VAR_OUTPUT
	EnO: BOOL;
	bDi_1: BOOL;
	bDi_2: BOOL;
	bDi_3: BOOL;
	bDi_4: BOOL;
	bDi_5: BOOL;
	bDi_6: BOOL;
	bDi_7: BOOL;
	bDi_8: BOOL;
	bDi_9: BOOL;
	bDi_10: BOOL;
	bDi_11: BOOL;
	bDi_12: BOOL;
	bDi_13: BOOL;
	bDi_14: BOOL;
	bDi_15: BOOL;
	bDi_16: BOOL;
	bError: BOOL;
END_VAR

VAR
	Channel_1_Input AT %I*: BOOL;
	Channel_2_Input AT %I*: BOOL;
	Channel_3_Input AT %I*: BOOL;
	Channel_4_Input AT %I*: BOOL;
	Channel_5_Input AT %I*: BOOL;
	Channel_6_Input AT %I*: BOOL;
	Channel_7_Input AT %I*: BOOL;
	Channel_8_Input AT %I*: BOOL;
	Channel_9_Input AT %I*: BOOL;
	Channel_10_Input AT %I*: BOOL;
	Channel_11_Input AT %I*: BOOL;
	Channel_12_Input AT %I*: BOOL;
	Channel_13_Input AT %I*: BOOL;
	Channel_14_Input AT %I*: BOOL;
	Channel_15_Input AT %I*: BOOL;
	Channel_16_Input AT %I*: BOOL;
	WcState_WcState AT %I*: BOOL;
	InfoData_State AT %I*: UINT;
	
	//FB-s
	EL1809_Error : FB_TerminalError;
END_VAR

EnO:=En;

//Error FB instance
EL1809_Error(
	En := TRUE,
	iTerminal_ID := iTerminal_ID,
	bWcState := WcState_WcState,
	uiInfoData_State := InfoData_State,
	pErrorSystem := ErrorSystem,
	bError => bError,
);

IF En THEN
	IF bError=FALSE THEN
		bDi_1:=Channel_1_Input;
		bDi_2:=Channel_2_Input;
		bDi_3:=Channel_3_Input;
		bDi_4:=Channel_4_Input;
		bDi_5:=Channel_5_Input;
		bDi_6:=Channel_6_Input;
		bDi_7:=Channel_7_Input;
		bDi_8:=Channel_8_Input;
		bDi_9:=Channel_9_Input;
		bDi_10:=Channel_10_Input;
		bDi_11:=Channel_11_Input;
		bDi_12:=Channel_12_Input;
		bDi_13:=Channel_13_Input;
		bDi_14:=Channel_14_Input;
		bDi_15:=Channel_15_Input;
		bDi_16:=Channel_16_Input;
	ELSE
		bDi_1:=FALSE;
		bDi_2:=FALSE;
		bDi_3:=FALSE;
		bDi_4:=FALSE;
		bDi_5:=FALSE;
		bDi_6:=FALSE;
		bDi_7:=FALSE;
		bDi_8:=FALSE;
		bDi_9:=FALSE;
		bDi_10:=FALSE;
		bDi_11:=FALSE;
		bDi_12:=FALSE;
		bDi_13:=FALSE;
		bDi_14:=FALSE;
		bDi_15:=FALSE;
		bDi_16:=FALSE;
	END_IF
END_IF

END_FUNCTION_BLOCK

// tc_mca_std_lib/POUs/Hardware/EtherCAT_Terminals/Digital_Inputs/EL1819
///EL1819 | HD EtherCAT Terminals, 16-channel digital input 24 V DC, 10 µs
FUNCTION_BLOCK EL1819

VAR_INPUT
	En: BOOL;
	iTerminal_ID : INT;
	ErrorSystem : POINTER TO ST_ErrorSystem;
END_VAR

VAR_OUTPUT
	EnO: BOOL;
	bDi_1: BOOL;
	bDi_2: BOOL;
	bDi_3: BOOL;
	bDi_4: BOOL;
	bDi_5: BOOL;
	bDi_6: BOOL;
	bDi_7: BOOL;
	bDi_8: BOOL;
	bDi_9: BOOL;
	bDi_10: BOOL;
	bDi_11: BOOL;
	bDi_12: BOOL;
	bDi_13: BOOL;
	bDi_14: BOOL;
	bDi_15: BOOL;
	bDi_16: BOOL;
	bError: BOOL;
END_VAR

VAR
	Channel_1_Input AT %I*: BOOL;
	Channel_2_Input AT %I*: BOOL;
	Channel_3_Input AT %I*: BOOL;
	Channel_4_Input AT %I*: BOOL;
	Channel_5_Input AT %I*: BOOL;
	Channel_6_Input AT %I*: BOOL;
	Channel_7_Input AT %I*: BOOL;
	Channel_8_Input AT %I*: BOOL;
	Channel_9_Input AT %I*: BOOL;
	Channel_10_Input AT %I*: BOOL;
	Channel_11_Input AT %I*: BOOL;
	Channel_12_Input AT %I*: BOOL;
	Channel_13_Input AT %I*: BOOL;
	Channel_14_Input AT %I*: BOOL;
	Channel_15_Input AT %I*: BOOL;
	Channel_16_Input AT %I*: BOOL;
	WcState_WcState AT %I*: BOOL;
	InfoData_State AT %I*: UINT;
	
	//FB-s
	EL1819_Error : FB_TerminalError;
END_VAR

EnO:=En;

//Error FB instance
EL1819_Error(
	En := TRUE,
	iTerminal_ID := iTerminal_ID,
	bWcState := WcState_WcState,
	uiInfoData_State := InfoData_State,
	pErrorSystem := ErrorSystem,
	bError => bError,
);

IF En THEN
	IF bError=FALSE THEN
		bDi_1:=Channel_1_Input;
		bDi_2:=Channel_2_Input;
		bDi_3:=Channel_3_Input;
		bDi_4:=Channel_4_Input;
		bDi_5:=Channel_5_Input;
		bDi_6:=Channel_6_Input;
		bDi_7:=Channel_7_Input;
		bDi_8:=Channel_8_Input;
		bDi_9:=Channel_9_Input;
		bDi_10:=Channel_10_Input;
		bDi_11:=Channel_11_Input;
		bDi_12:=Channel_12_Input;
		bDi_13:=Channel_13_Input;
		bDi_14:=Channel_14_Input;
		bDi_15:=Channel_15_Input;
		bDi_16:=Channel_16_Input;
	ELSE
		bDi_1:=FALSE;
		bDi_2:=FALSE;
		bDi_3:=FALSE;
		bDi_4:=FALSE;
		bDi_5:=FALSE;
		bDi_6:=FALSE;
		bDi_7:=FALSE;
		bDi_8:=FALSE;
		bDi_9:=FALSE;
		bDi_10:=FALSE;
		bDi_11:=FALSE;
		bDi_12:=FALSE;
		bDi_13:=FALSE;
		bDi_14:=FALSE;
		bDi_15:=FALSE;
		bDi_16:=FALSE;
	END_IF
END_IF

END_FUNCTION_BLOCK

// tc_mca_std_lib/POUs/Hardware/EtherCAT_Terminals/Digital_Inputs/FB_EL1252ASM_v1_00
FUNCTION_BLOCK FB_EL1252ASM_v1_00
VAR_INPUT
	En: BOOL;
END_VAR
VAR_OUTPUT
	EnO: BOOL;
	Di_1: BOOL;
	Di_2: BOOL;
	Di_1_LatchTimePos: ULINT;
	Di_2_LatchTimePos: ULINT;
	Di_1_LatchTimeNeg: ULINT;
	Di_2_LatchTimeNeg: ULINT;
	///Below bits can be used but then they must be enabled in the COE of the card. Nicklas suggested to not use these (since something wss written that you then only were allowed to read the latch time onece (some kkind of auto reset??))	
	///Di_1_LatchNeg:BOOL;
	///	Di_1_LatchPos:BOOL;
	///	Di_2_LatchNeg:BOOL;
	///	Di_2_LatchPos:BOOL;
	Error: BOOL;
END_VAR
VAR
	Channel_1_Input AT %I*: BOOL;
	Channel_2_Input AT %I*: BOOL;
	///Latch_Status1 AT %I*: USINT;
	///	Latch_Status2 AT %I*: USINT;
	Latch_LatchPos1 AT %I*: ULINT;
	Latch_LatchNeg1 AT %I*: ULINT;
	Latch_LatchPos2 AT %I*: ULINT;
	Latch_LatchNeg2 AT %I*: ULINT;
	WcState_WcState AT %I*: BOOL;
	InfoData_State AT %I*: UINT;
END_VAR

EnO:=En;

IF En AND (WcState_WcState OR InfoData_State<>16#8) THEN //InfoData_State==0 => in OP mode
	Error:=TRUE;
ELSE
	Error:=FALSE;
END_IF

IF En THEN
	IF Error=FALSE THEN
		Di_1:=Channel_1_Input;
		Di_2:=Channel_2_Input;
	(*	Di_1_LatchPos:=Latch_Status1.0;
		Di_1_LatchNeg:=Latch_Status1.1;
		Di_2_LatchPos:=Latch_Status2.0;
		Di_2_LatchNeg:=Latch_Status2.1;*)
		Di_1_LatchTimePos:=Latch_LatchPos1;
		Di_2_LatchTimePos:=Latch_LatchPos2;		
		Di_1_LatchTimeNeg:=Latch_LatchNeg1;		
		Di_2_LatchTimeNeg:=Latch_LatchNeg2;
		
	ELSE
		Di_1:=FALSE;
		Di_2:=FALSE;
	END_IF
END_IF

END_FUNCTION_BLOCK

// tc_mca_std_lib/POUs/Hardware/EtherCAT_Terminals/Digital_Outputs/EL2014
FUNCTION_BLOCK EL2014
VAR_INPUT
	En: BOOL;
	iTerminal_ID : INT; 
	bDo_1: BOOL;
	bDo_2: BOOL;
	bDo_3: BOOL;
	bDo_4: BOOL;
	ErrorSystem : POINTER TO ST_ErrorSystem;
END_VAR

VAR_OUTPUT
	EnO : BOOL;
	bError : BOOL;
END_VAR

VAR
	Channel_1_Output AT %Q*: BOOL;
	Channel_2_Output AT %Q*: BOOL;
	Channel_3_Output AT %Q*: BOOL;
	Channel_4_Output AT %Q*: BOOL;
	WcState_WcState AT %I*: BOOL;
	InfoData_State AT %I*: UINT;
	
	//FB-s
	EL2014_Error : FB_TerminalError;
END_VAR

(*
* TODO:
* Channel diagnostic variables and device diag variables
*)

EnO:=En;

EL2014_Error(
	En := TRUE,
	iTerminal_ID := iTerminal_ID,
	bWcState := WcState_WcState,
	uiInfoData_State := InfoData_State,
	pErrorSystem := ErrorSystem,
	bError => bError,
);

IF En THEN
	IF bError=FALSE THEN
		Channel_1_Output:=bDo_1;
		Channel_2_Output:=bDo_2;
		Channel_3_Output:=bDo_3;
		Channel_4_Output:=bDo_4;
	ELSE
		Channel_1_Output:=FALSE;
		Channel_2_Output:=FALSE;
		Channel_3_Output:=FALSE;
		Channel_4_Output:=FALSE;
	END_IF
END_IF

END_FUNCTION_BLOCK

// tc_mca_std_lib/POUs/Hardware/EtherCAT_Terminals/Digital_Outputs/EL2252
///EL2252 | XFC, 2-channel digital output terminal with time stamp, tri-state
FUNCTION_BLOCK EL2252
VAR_INPUT
	En: BOOL;
	iTerminal_ID : INT; 
	bDo_1: BOOL;
	bDo_2: BOOL;
ErrorSystem : POINTER TO ST_ErrorSystem;
END_VAR

VAR_OUTPUT
	EnO : BOOL;
	bError : BOOL;
END_VAR

VAR
	Channel_1_Output AT %Q*: BOOL;
	Channel_2_Output AT %Q*: BOOL;
	WcState_WcState AT %I*: BOOL;
	InfoData_State AT %I*: UINT;
	
	//FB-s
	EL2252_Error : FB_TerminalError;
END_VAR

(*
* TODO:
* Add the DC sync variables
*)

EL2252_Error(
	En := TRUE,
	iTerminal_ID := iTerminal_ID,
	bWcState := WcState_WcState,
	uiInfoData_State := InfoData_State,
	pErrorSystem := ErrorSystem,
	bError => bError,
);

IF En THEN
	IF bError=FALSE THEN
		Channel_1_Output:=bDo_1;
		Channel_2_Output:=bDo_2;
	ELSE
		Channel_1_Output:=FALSE;
		Channel_2_Output:=FALSE;
	END_IF
END_IF

END_FUNCTION_BLOCK

// tc_mca_std_lib/POUs/Hardware/EtherCAT_Terminals/Digital_Outputs/EL2808
FUNCTION_BLOCK EL2808

VAR_INPUT
	En: BOOL;
	iTerminal_ID : INT; 
	bDo_1: BOOL;
	bDo_2: BOOL;
	bDo_3: BOOL;
	bDo_4: BOOL;
	bDo_5: BOOL;
	bDo_6: BOOL;
	bDo_7: BOOL;
	bDo_8: BOOL;
	ErrorSystem : POINTER TO ST_ErrorSystem;
END_VAR

VAR_OUTPUT
	EnO : BOOL;
	bError : BOOL;
END_VAR

VAR
	Channel_1_Output AT %Q*: BOOL;
	Channel_2_Output AT %Q*: BOOL;
	Channel_3_Output AT %Q*: BOOL;
	Channel_4_Output AT %Q*: BOOL;
	Channel_5_Output AT %Q*: BOOL;
	Channel_6_Output AT %Q*: BOOL;
	Channel_7_Output AT %Q*: BOOL;
	Channel_8_Output AT %Q*: BOOL;
	WcState_WcState AT %I*: BOOL;
	InfoData_State AT %I*: UINT;
	
	//FB-s
	EL2808_Error : FB_TerminalError;
END_VAR

EnO:=En;

EL2808_Error(
	En := TRUE,
	iTerminal_ID := iTerminal_ID,
	bWcState := WcState_WcState,
	uiInfoData_State := InfoData_State,
	pErrorSystem := ErrorSystem,
	bError => bError,
);

IF En THEN
	IF bError=FALSE THEN
		Channel_1_Output:=bDo_1;
		Channel_2_Output:=bDo_2;
		Channel_3_Output:=bDo_3;
		Channel_4_Output:=bDo_4;
		Channel_5_Output:=bDo_5;
		Channel_6_Output:=bDo_6;
		Channel_7_Output:=bDo_7;
		Channel_8_Output:=bDo_8;
	ELSE
		Channel_1_Output:=FALSE;
		Channel_2_Output:=FALSE;
		Channel_3_Output:=FALSE;
		Channel_4_Output:=FALSE;
		Channel_5_Output:=FALSE;
		Channel_6_Output:=FALSE;
		Channel_7_Output:=FALSE;
		Channel_8_Output:=FALSE;
	END_IF
END_IF

END_FUNCTION_BLOCK

// tc_mca_std_lib/POUs/Hardware/EtherCAT_Terminals/Digital_Outputs/EL2819
FUNCTION_BLOCK EL2819
VAR_INPUT
	En: BOOL;
	iTerminal_ID : INT; 
	bDo_1: BOOL;
	bDo_2: BOOL;
	bDo_3: BOOL;
	bDo_4: BOOL;
	bDo_5: BOOL;
	bDo_6: BOOL;
	bDo_7: BOOL;
	bDo_8: BOOL;
	bDo_9: BOOL;
	bDo_10: BOOL;
	bDo_11: BOOL;
	bDo_12: BOOL;
	bDo_13: BOOL;
	bDo_14: BOOL;
	bDo_15: BOOL;
	bDo_16: BOOL;
	ErrorSystem : POINTER TO ST_ErrorSystem;
END_VAR

VAR_OUTPUT
	EnO : BOOL;
	bError : BOOL;
END_VAR

VAR
	Channel_1_Output AT %Q*: BOOL;
	Channel_2_Output AT %Q*: BOOL;
	Channel_3_Output AT %Q*: BOOL;
	Channel_4_Output AT %Q*: BOOL;
	Channel_5_Output AT %Q*: BOOL;
	Channel_6_Output AT %Q*: BOOL;
	Channel_7_Output AT %Q*: BOOL;
	Channel_8_Output AT %Q*: BOOL;
	Channel_9_Output AT %Q*: BOOL;
	Channel_10_Output AT %Q*: BOOL;
	Channel_11_Output AT %Q*: BOOL;
	Channel_12_Output AT %Q*: BOOL;
	Channel_13_Output AT %Q*: BOOL;
	Channel_14_Output AT %Q*: BOOL;
	Channel_15_Output AT %Q*: BOOL;
	Channel_16_Output AT %Q*: BOOL;
	
	WcState_WcState AT %I*: BOOL;
	InfoData_State AT %I*: UINT;
	
	//FB-s
	EL2819_Error : FB_TerminalError;
END_VAR

(*
* TODO:
* Channel diagnostic variables and device diag variables
*)

EnO:=En;

EL2819_Error(
	En := TRUE,
	iTerminal_ID := iTerminal_ID,
	bWcState := WcState_WcState,
	uiInfoData_State := InfoData_State,
	pErrorSystem := ErrorSystem,
	bError => bError,
);

IF En THEN
	IF bError=FALSE THEN
		Channel_1_Output:=bDo_1;
		Channel_2_Output:=bDo_2;
		Channel_3_Output:=bDo_3;
		Channel_4_Output:=bDo_4;
		Channel_5_Output:=bDo_5;
		Channel_6_Output:=bDo_6;
		Channel_7_Output:=bDo_7;
		Channel_8_Output:=bDo_8;
		Channel_9_Output:=bDo_9;
		Channel_10_Output:=bDo_10;
		Channel_11_Output:=bDo_11;
		Channel_12_Output:=bDo_12;
		Channel_13_Output:=bDo_13;
		Channel_14_Output:=bDo_14;
		Channel_15_Output:=bDo_15;
		Channel_16_Output:=bDo_16;
	ELSE
		Channel_1_Output:=FALSE;
		Channel_2_Output:=FALSE;
		Channel_3_Output:=FALSE;
		Channel_4_Output:=FALSE;
		Channel_5_Output:=FALSE;
		Channel_6_Output:=FALSE;
		Channel_7_Output:=FALSE;
		Channel_8_Output:=FALSE;
		Channel_9_Output:=FALSE;
		Channel_10_Output:=FALSE;
		Channel_11_Output:=FALSE;
		Channel_12_Output:=FALSE;
		Channel_13_Output:=FALSE;
		Channel_14_Output:=FALSE;
		Channel_15_Output:=FALSE;
		Channel_16_Output:=FALSE;
	END_IF
END_IF

END_FUNCTION_BLOCK

// tc_mca_std_lib/POUs/Hardware/EtherCAT_Terminals/Measuring_Terminals/EL5002
//EL5002 | 2-chennel SSI absolute encoder terminal
FUNCTION_BLOCK EL5002

VAR_INPUT
	En: BOOL;
	iTerminal_ID : INT;
	ErrorSystem : POINTER TO ST_ErrorSystem;
END_VAR

VAR_OUTPUT
	EnO: BOOL;
	Ch1_Counter_Value : UDINT;
	Ch2_Counter_Value : UDINT;
	bError: BOOL;
END_VAR

VAR
	udi_Ch1_Cnt_Value AT %I* : UDINT;
	udi_Ch2_Cnt_Value AT %I* : UDINT;
	WcState_WcState AT %I*: BOOL;
	InfoData_State AT %I*: UINT;
	
	//FB-s
	EL5002_Error : FB_TerminalError;
END_VAR

(*
* TODO:
* Channel Status words
*)

EnO:=En;

//Error FB instance
EL5002_Error(
	En := TRUE,
	iTerminal_ID := iTerminal_ID,
	bWcState := WcState_WcState,
	uiInfoData_State := InfoData_State,
	pErrorSystem := ErrorSystem,
	bError => bError,
);

IF EN THEN
	IF NOT bError THEN
		Ch1_Counter_Value := udi_Ch1_Cnt_Value;
		Ch2_Counter_Value := udi_Ch2_Cnt_Value;
	ELSE
		Ch1_Counter_Value := 0;
		Ch2_Counter_Value := 0;
	END_IF
END_IF

END_FUNCTION_BLOCK

// tc_mca_std_lib/POUs/Hardware/EtherCAT_Terminals/Measuring_Terminals/EL5021
//EL5021 | 1-channel Sin/Cos encoder
FUNCTION_BLOCK EL5021

VAR_INPUT
	En: BOOL;
	iTerminal_ID : INT;
	ErrorSystem : POINTER TO ST_ErrorSystem;
END_VAR

VAR_OUTPUT
	EnO: BOOL;
	Counter_Value : UDINT;
	Latch_Value : UDINT;
	bError: BOOL;
END_VAR

VAR
	udiCounter_Value AT %I* : UDINT;
	udiLatch_Value AT %I* : UDINT;
	WcState_WcState AT %I*: BOOL;
	InfoData_State AT %I*: UINT;
	
	//FB-s
	EL5021_Error : FB_TerminalError;
END_VAR

(*
* TODO:
* Channel Status words, control words
*)

EnO:=En;

//Error FB instance
EL5021_Error(
	En := TRUE,
	iTerminal_ID := iTerminal_ID,
	bWcState := WcState_WcState,
	uiInfoData_State := InfoData_State,
	pErrorSystem := ErrorSystem,
	bError => bError,
);

IF EN THEN
	IF NOT bError THEN
		Counter_Value := udiCounter_Value;
		Latch_Value := udiLatch_Value;
	ELSE
		Counter_Value := 0;
		Latch_Value := 0;
	END_IF
END_IF

END_FUNCTION_BLOCK

// tc_mca_std_lib/POUs/Hardware/EtherCAT_Terminals/Measuring_Terminals/EL5042
//EL5042 | 2-channel BiSS-C absolute encoder terminal
FUNCTION_BLOCK EL5042

VAR_INPUT
	En: BOOL;
	iTerminal_ID : INT;
	ErrorSystem : POINTER TO ST_ErrorSystem;
END_VAR

VAR_OUTPUT
	EnO: BOOL;
	Ch1_Position : ULINT;
	Ch2_Position : ULINT;
	bError: BOOL;
END_VAR

VAR
	FB_Inputs_ch1_Position AT %I* : ULINT;
	FB_Inputs_ch2_Position AT %I* : ULINT;
	WcState_WcState AT %I*: BOOL;
	InfoData_State AT %I*: UINT;
	
	//FB-s
	EL5042_Error : FB_TerminalError;
END_VAR

(*
* TODO:
* Channel Status words
*)

EnO:=En;

//Error FB instance
EL5042_Error(
	En := TRUE,
	iTerminal_ID := iTerminal_ID,
	bWcState := WcState_WcState,
	uiInfoData_State := InfoData_State,
	pErrorSystem := ErrorSystem,
	bError => bError,
);

IF EN THEN
	IF NOT bError THEN
		Ch1_Position := FB_Inputs_ch1_Position;
		Ch2_Position := FB_Inputs_ch2_Position;
	ELSE
		Ch1_Position := 0;
		Ch2_Position := 0;
	END_IF
END_IF

END_FUNCTION_BLOCK

// tc_mca_std_lib/POUs/Hardware/EtherCAT_Terminals/Measuring_Terminals/EL5101
// EL5101 | 1-channel incremental encoder terminal, 5V, RS422
FUNCTION_BLOCK EL5101

VAR_INPUT
	En: BOOL;
	iTerminal_ID : INT;
	ErrorSystem : POINTER TO ST_ErrorSystem;
END_VAR

VAR_OUTPUT
	EnO: BOOL;
	Counter_Value : UINT;
	Latch_Value : UINT;
	bError: BOOL;
END_VAR

VAR
	uiCounter_Value AT %I* : UINT;
	uiLatch_Value AT %I* : UINT;
	WcState_WcState AT %I*: BOOL;
	InfoData_State AT %I*: UINT;
	
	//FB-s
	EL5101_Error : FB_TerminalError;
END_VAR

(*
* TODO:
* Channel Status word, control words
*)

EnO:=En;

//Error FB instance
EL5101_Error(
	En := TRUE,
	iTerminal_ID := iTerminal_ID,
	bWcState := WcState_WcState,
	uiInfoData_State := InfoData_State,
	pErrorSystem := ErrorSystem,
	bError => bError,
);

IF EN THEN
	IF NOT bError THEN
		Counter_Value := uiCounter_Value;
		Latch_Value := uiLatch_Value;
	ELSE
		Counter_Value := 0;
		Latch_Value := 0;
	END_IF
END_IF

END_FUNCTION_BLOCK

// tc_mca_std_lib/POUs/Hardware/EtherCAT_Terminals/Motion/EL7211_v1_00
///EL7211 | Servo motor termional 5 A
FUNCTION_BLOCK EL7211_v1_00
VAR_INPUT
	En: BOOL;
END_VAR
VAR_OUTPUT
	EnO: BOOL;

	bError: BOOL;
END_VAR
VAR
	WcState_WcState AT %I*: BOOL;
	InfoData_State AT %I*: UINT;
END_VAR

EnO:=En;

IF En AND (WcState_WcState OR InfoData_State<>16#8) THEN
	bError:=TRUE;
ELSE
	bError:=FALSE;
END_IF

END_FUNCTION_BLOCK

// tc_mca_std_lib/POUs/Hardware/EtherCAT_Terminals/Motion/EL9576_v1_00
///EL9576 | Brake terminal (vap and resistor)
FUNCTION_BLOCK EL9576_v1_00
VAR_INPUT
	En: BOOL;
END_VAR
VAR_OUTPUT
	EnO: BOOL;
	bError: BOOL;	
	OverTemperature: BOOL;
	I2TError : BOOL;
	I2TWarning : BOOL;
	OverVoltage  : BOOL;
	UnderVoltage : BOOL;
	ChopperOn : BOOL;
	DCLinkVoltage : LREAL;
	DutyCycle  : LREAL;
	ResistorCurrent : LREAL;
	
END_VAR
VAR
	BCTOverTemperature AT %I*: BOOL;
	BCTI2TError AT %I*: BOOL;
	BCTI2TWarning AT %I*: BOOL;
	BCTOverVoltage  AT %I*: BOOL;
	BCTUnderVoltage  AT %I*: BOOL;
	BCTChopperOn  AT %I*: BOOL;
	BCTDCLinkVoltage AT %I*: UDINT;
	BCTDutyCycle  AT %I*: USINT;
	BCTResistorCurrent AT %I*: UDINT;
	WcState_WcState AT %I*: BOOL;
	InfoData_State AT %I*: UINT;
	
END_VAR

EnO:=En;

IF En AND (WcState_WcState OR InfoData_State<>16#8 OR BCTI2TError OR BCTI2TWarning OR BCTOverTemperature OR BCTOverVoltage OR BCTUnderVoltage) THEN
	bError:=TRUE;
ELSE
	bError:=FALSE;
END_IF

OverTemperature:=BCTOverTemperature;
I2TError:=BCTI2TError;
I2TWarning:=BCTI2TWarning;
OverVoltage:=BCTOverVoltage;
UnderVoltage:=bctUnderVoltage;
ChopperOn:=bctChopperOn;
DCLinkVoltage:=UDINT_TO_LREAL(bctDCLinkVoltage);
DutyCycle:=USINT_TO_LREAL(BCTDutyCycle);
ResistorCurrent:=UDINT_TO_LREAL(BCTResistorCurrent);

END_FUNCTION_BLOCK

// tc_mca_std_lib/POUs/Hardware/EtherCAT_Terminals/System/EL9410
//EL9410 | E-Bus power supplier and refresher, diagnostics
FUNCTION_BLOCK EL9410

VAR_INPUT
	En: BOOL;
	iTerminal_ID : INT;
	ErrorSystem : POINTER TO ST_ErrorSystem;
END_VAR

VAR_OUTPUT
	EnO: BOOL;
	bError: BOOL;
END_VAR

VAR
	bStatus_Us_UV AT %I* : BOOL;
	bStatus_Up_UV AT %I* : BOOL;
	WcState_WcState AT %I*: BOOL;
	InfoData_State AT %I*: UINT;
	
	//FB-s
	EL9410_Error : FB_TerminalError;
END_VAR

(*
* TODO:
* Status bits
*)

EnO:=En;

//Error FB instance
EL9410_Error(
	En := TRUE,
	iTerminal_ID := iTerminal_ID,
	bWcState := WcState_WcState,
	uiInfoData_State := InfoData_State,
	pErrorSystem := ErrorSystem,
	bError => bError,
);

END_FUNCTION_BLOCK

// tc_mca_std_lib/POUs/Hardware/EtherCAT_Terminals/System/EL9505
//EL9505 | Power supply terminal 5V
FUNCTION_BLOCK EL9505

VAR_INPUT
	En: BOOL;
	iTerminal_ID : INT;
	ErrorSystem : POINTER TO ST_ErrorSystem;
END_VAR

VAR_OUTPUT
	EnO: BOOL;
	bError: BOOL;
END_VAR

VAR
	bStatus_Uo_Power_OK AT %I* : BOOL;
	bStatus_Uo_Overload AT %I* : BOOL;
	WcState_WcState AT %I*: BOOL;
	InfoData_State AT %I*: UINT;
	
	//FB-s
	EL9505_Error : FB_TerminalError;
END_VAR

(*
* TODO:
* Status bits
*)
EnO:=En;

//Error FB instance
EL9505_Error(
	En := TRUE,
	iTerminal_ID := iTerminal_ID,
	bWcState := WcState_WcState,
	uiInfoData_State := InfoData_State,
	pErrorSystem := ErrorSystem,
	bError => bError,
);

END_FUNCTION_BLOCK

// tc_mca_std_lib/POUs/Hardware/Other/EK1200
FUNCTION_BLOCK EK1200
VAR_INPUT
	En: BOOL;
END_VAR
VAR_OUTPUT
	EnO: BOOL;
END_VAR

EnO:=En;

END_FUNCTION_BLOCK

// tc_mca_std_lib/POUs/Motion/FB_NcAxis
///#########################################################
///Function block to communicate between Nc and Plc.
///
///	Library:		
///	Tc2_MC2.lib
///
///	Global Variables:
///	
///	Data types:
///	
///	External functions:
///
///###########################################################
FUNCTION_BLOCK FB_NcAxis
VAR
	sVersion: STRING:='1.0.0';
END_VAR
VAR_INPUT
	En: BOOL;
END_VAR
VAR_OUTPUT
	EnO: BOOL;
	bError: BOOL;
	Status: ST_AxisStatus;
END_VAR
VAR
	Axis: AXIS_REF;
	InfoData_State AT %I*: UINT;
END_VAR

EnO:=En;

IF En AND InfoData_State<>16#8 THEN
	bError:=TRUE;
ELSE
	bError:=FALSE;
END_IF

IF En THEN
	Axis.ReadStatus();
	Status:=Axis.Status;
END_IF

END_FUNCTION_BLOCK

// Tests/Helpers/FB_CauseNCError
FUNCTION_BLOCK FB_CauseNCError
(*
    Simulate an NC error.
    This will look like a real NC error for everyone, including TwinCAT itself.
*)
VAR_IN_OUT
    Axis: AXIS_REF;
END_VAR
VAR_INPUT
    bExecute: BOOL;
    nErrorCode: UDINT;
END_VAR
VAR_OUTPUT
    bBusy: BOOL;
    bDone: BOOL;
END_VAR
VAR
    rtExec: R_TRIG;
    adsWrite: ADSWRITE;
    mcReadDriveAddress: MC_ReadDriveAddress;
END_VAR


rtExec(CLK:=bExecute);
IF NOT bExecute THEN
    bDone := FALSE;
END_IF
IF rtExec.Q THEN
    bBusy := TRUE;
END_IF
IF bBusy AND NOT mcReadDriveAddress.Done THEN
    mcReadDriveAddress(
        Axis:=Axis,
        Execute:=TRUE,
        DriveAddress=>Axis.DriveAddress);
END_IF
IF bBusy AND mcReadDriveAddress.Done THEN
    bBusy := TRUE;
    adsWrite(
        PORT:=501,
        IDXGRP:=16#4200 + Axis.DriveAddress.NcDriveId,
        IDXOFFS:=16#0019,
        LEN:=SIZEOF(nErrorCode),
        SRCADDR:=ADR(nErrorCode),
        WRITE:=TRUE,
        BUSY=>bBusy);
    IF NOT bBusy THEN
        bDone := TRUE;
        adsWrite(WRITE:=FALSE);
    END_IF
END_IF

END_FUNCTION_BLOCK

// Tests/Helpers/FB_MotorTestSuite
FUNCTION_BLOCK FB_MotorTestSuite EXTENDS TcUnit.FB_TestSuite
(*
    Base class for motion tests.

    Contains some helper methods that would otherwise need to be instantiated many times,
    but in this form can be accessed quickly and succinctly in the test suite.
*)

METHOD SetEnables
(*
    Set a motion stage's enables such that it is fully allowed to move.
*)
VAR_IN_OUT
    stMotionStage: ST_MotionStage;
END_VAR
stMotionStage.bHardwareEnable := TRUE;
stMotionStage.bLimitBackwardEnable := TRUE;
stMotionStage.bLimitForwardEnable := TRUE;
stMotionStage.bPowerSelf := TRUE;
END_METHOD

METHOD SetEnablesPMPS
(*
    Set a motion stage's enables such that only PMPS would be preventing a move.
*)
VAR_IN_OUT
    stMotionStage: ST_MotionStage;
END_VAR

SetEnables(stMotionStage);
stMotionStage.bPowerSelf := FALSE;
END_METHOD

METHOD SetGoodState
(*
    Mark a state as valid and ready to use.
*)
VAR_IN_OUT
    stPositionState: ST_PositionState;
END_VAR
stPositionState.bMoveOk := TRUE;
stPositionState.bValid := TRUE;
END_METHOD

END_FUNCTION_BLOCK

// Tests/Helpers/FB_PMPSJsonTestHelper
FUNCTION_BLOCK FB_PMPSJsonTestHelper
(*
    Create a JSON doc in memory to match the input structs
    Assumes 1 device for simplicity
    Writes to the global pmps json doc
*)
VAR_IN_OUT
    astBeamParams: ARRAY[*] OF ST_DbStateParams;
END_VAR
VAR_INPUT
    bExecute: BOOL;
    sDevName: STRING;
END_VAR
VAR_OUTPUT
END_VAR
VAR
    rtExec: R_TRIG;
    jsonRoot: SJsonValue;
    jsonDevice: SJsonValue;
    ajsonState: ARRAY[0..GeneralConstants.MAX_STATES] OF SJsonValue;
    fbJson: FB_JsonDomParser;

    nIter: DINT;
    nId: DINT;

    aseVRange: ARRAY[0..GeneralConstants.MAX_STATES] OF STRING;
    asRate: ARRAY[0..GeneralConstants.MAX_STATES] OF STRING;
    asBCRange: ARRAY[0..GeneralConstants.MAX_STATES] OF STRING;
    asTran: ARRAY[0..GeneralConstants.MAX_STATES] OF STRING;
END_VAR


rtExec(CLK:=bExecute);
IF NOT rtExec.Q THEN
    RETURN;
END_IF

jsonRoot := fbJson.NewDocument();
jsonDevice := fbJson.AddObjectMember(jsonRoot, sDevName);
FOR nIter := LOWER_BOUND(astBeamParams, 1) TO UPPER_BOUND(astBeamParams, 1) DO
    ajsonState[nIter] := fbJson.AddObjectMember(jsonDevice, astBeamParams[nIter].sPmpsState);

    nId := nId + 1;
    fbJson.AddIntMember(
        v:=ajsonState[nIter],
        member:='id',
        value:=nId,
    );
    fbJson.AddStringMember(
        v:=ajsonState[nIter],
        member:='beamline',
        value:='tst',
    );
    aseVRange[nIter] := bitmaskToString(astBeamParams[nIter].stBeamParams.neVRange, 32);
    fbJson.AddStringMember(
        v:=ajsonState[nIter],
        member:='neVRange',
        value:=aseVRange[nIter],
    );
    asRate[nIter] := UDINT_TO_STRING(astBeamParams[nIter].stBeamParams.nRate);
    fbJson.AddStringMember(
        v:=ajsonState[nIter],
        member:='nRate',
        value:=asRate[nIter],
    );
    fbJson.AddStringMember(
        v:=ajsonState[nIter],
        member:='ap_ygap',
        value:='',
    );
    fbJson.AddStringMember(
        v:=ajsonState[nIter],
        member:='ap_xgap',
        value:='',
    );
    fbJson.AddStringMember(
        v:=ajsonState[nIter],
        member:='damage_limit',
        value:='',
    );
    fbJson.AddStringMember(
        v:=ajsonState[nIter],
        member:='notes',
        value:='',
    );
    fbJson.AddStringMember(
        v:=ajsonState[nIter],
        member:='reactive_temp',
        value:='',
    );
    fbJson.AddStringMember(
        v:=ajsonState[nIter],
        member:='reactive_pressure',
        value:='',
    );
    asBCRange[nIter] := bitmaskToString(astBeamParams[nIter].stBeamParams.nBCRange, 15);
    fbJson.AddStringMember(
        v:=ajsonState[nIter],
        member:='nBeamClassRange',
        value:=asBCRange[nIter],
    );
    fbJson.AddStringMember(
        v:=ajsonState[nIter],
        member:='name',
        value:=astBeamParams[nIter].sPmpsState,
    );
    asTran[nIter] := REAL_TO_STRING(astBeamParams[nIter].stBeamParams.nTran);
    fbJson.AddStringMember(
        v:=ajsonState[nIter],
        member:='nTran',
        value:=asTran[nIter],
    );
    fbJson.AddStringMember(
        v:=ajsonState[nIter],
        member:='ap_name',
        value:='None',
    );
    fbJson.AddStringMember(
        v:=ajsonState[nIter],
        member:='ap_ycenter',
        value:='',
    );
    fbJson.AddStringMember(
        v:=ajsonState[nIter],
        member:='ap_xcenter',
        value:='',
    );
    fbJson.AddStringMember(
        v:=ajsonState[nIter],
        member:='pulse_energy',
        value:='',
    );
    fbJson.AddBoolMember(
        v:=ajsonState[nIter],
        member:='special',
        value:=FALSE,
    );
END_FOR

PMPS_GVL.BP_jsonDoc := jsonRoot;

METHOD bitmaskToString : STRING
VAR_INPUT
    nBitmask: DWORD;
    nBits: UINT;
END_VAR
VAR
    nIter: UINT;
END_VAR

bitmaskToString := '';
FOR nIter := 1 TO nBits DO
    bitmaskToString := CONCAT(DWORD_TO_STRING(SHR(nBitmask, nIter - 1) AND 1), bitmaskToString);
END_FOR
END_METHOD

END_FUNCTION_BLOCK

// Tests/Helpers/FB_TestHelperSetAndMove
FUNCTION_BLOCK FB_TestHelperSetAndMove
(*
    Set an stMotionStage to a start position, then cause a move.
    On rising edge of bExecute, errors are cleared, the user enable is set to FALSE, and the position is set.
    After the position is set, user enable is re-introduced and a move begins.

    The progress of this function block for the purposes of a unit test can be monitored via the outputs.

    The motion stage should have its own FB_MotionStage or some stand-in for it running on outside of the FB.

    This is, in itself, tested in FB_TestHelperSetAndMove_Test.
*)
VAR_IN_OUT
    // The motion state to test with
    stMotionStage: ST_MotionStage;
END_VAR
VAR_INPUT
    // Begin on rising edge, stop on falling edge.
    bExecute: BOOL;
    // The position to set the motor to
    fStartPosition: LREAL;
    // The goal to move the motor towards
    fGoalPosition: LREAL;
    // The velocity to move at
    fVelocity: LREAL;
    // If TRUE, we'll set all the hardware enable signals. Leave this as FALSE if your testing involves any of the hardware enables.
    bHWEnable: BOOL;
END_VAR
VAR_OUTPUT
    // Goes to TRUE once the motor has no errors and is deactivated.
    bResetDone: BOOL;
    // Goes to TRUE once the set position completes.
    bSetDone: BOOL;
    // Goes to TRUE once the motor begins moving.
    bMotionStarted: BOOL;
    // Goes to TRUE once the motor reaches its destination.
    bMoveDone: BOOL;
    // If bBusy is FALSE, the function block is ready for a new request. Goes to TRUE after bExecute rises and back to FALSE after bMoveDone or bError rises. Also goes to FALSE after the motor stops following bExecute being dropped to FALSE.
    bBusy: BOOL;
    // Goes to TRUE in case of an error from FB_MotionRequest
    bError: BOOL;
    // Counts up from bExecute's rising trigger. Can be used to implement a timeout.
    tElapsed: TIME;
    // Current motor position in case you're looking for it
    fActPosition: LREAL;
    // Goes to TRUE if we're trying to stop a move. We'll stop an in-progress move when bExecute goes to FALSE, and we'll make sure the motor fully stops before responding to the next bExecute rising edge.
    bStoppingMotor: BOOL;
END_VAR
VAR
    fbMoveRequest: FB_MotionRequest;
    mcSetPos: MC_SetPosition;
    tonTimeout: TON;
    rtExec: R_TRIG;
    ftExec: F_TRIG;
    bExecQueued: BOOL;
    nLatchError: UDINT;
END_VAR


tonTimeout(
    IN:=bExecute,
    PT:=T#1h,
    ET=>tElapsed,
);
rtExec(CLK:=bExecute);
ftExec(CLK:=bExecute);

// Set the outputs to known values on exec
bResetDone R= rtExec.Q;
bSetDone R= rtExec.Q;
bMotionStarted R= rtExec.Q;
bMoveDone R= rtExec.Q;
bBusy S= rtExec.Q;
bError R= rtExec.Q;

bExecQueued S= rtExec.Q;
bExecQueued R= ftExec.Q;
bStoppingMotor S= ftExec.Q;

// Set the hardware enables if asked
IF bHWEnable THEN
    stMotionStage.bLimitForwardEnable := TRUE;
    stMotionStage.bLimitBackwardEnable := TRUE;
    stMotionStage.bHardwareEnable := TRUE;
    stMotionStage.bPowerSelf := TRUE;
END_IF


// Note that we only reset if it's needed, e.g. the motor has an error or is enabled or moving etc. etc.
bResetDone S= stMotionStage.bError = FALSE AND stMotionStage.bBusy = FALSE AND stMotionStage.bAllEnable = FALSE;

// All uses of fbMoveRequest are in this IF/ELSE tree
IF bStoppingMotor THEN
    // Continue stopping the motor from previous cycles
    fbMoveRequest(
        stMotionStage:=stMotionStage,
        bExecute:=FALSE,
    );
    stMotionStage.bExecute := FALSE;
    bStoppingMotor R= NOT stMotionStage.Axis.Status.ControlLoopClosed AND NOT fbMoveRequest.bBusy;
ELSIF bExecQueued THEN
    // First exec cycle: bring these to FALSE for later use
    bExecQueued := FALSE;
    stMotionStage.bUserEnable := FALSE;
    fbMoveRequest(
        stMotionStage:=stMotionStage,
        bExecute:=FALSE,
        bReset:=FALSE,
    );
ELSIF NOT bResetDone THEN
    // Other cycles: reset until we're done resetting
    fbMoveRequest(
        stMotionStage:=stMotionStage,
        bReset:=bExecute,
    );
ELSIF fStartPosition <> fGoalPosition THEN
    // Later: do the move
    // Important to not enable the motor until the set position is done
    stMotionStage.bUserEnable := bSetDone;
    fbMoveRequest(
        stMotionStage:=stMotionStage,
        bExecute:=bSetDone AND bExecute AND NOT bMoveDone AND NOT bError,
        bReset:=FALSE,
        enumMotionRequest:=E_MotionRequest.INTERRUPT,
        fPos:=fGoalPosition,
        fVel:=fVelocity,
    );
    bMotionStarted S= bSetDone AND fbMoveRequest.bExecute AND stMotionStage.bBusy AND stMotionStage.stAxisStatus.fActPosition <> fStartPosition;
    bMoveDone S= bMotionStarted AND stMotionStage.stAxisStatus.fActPosition = fGoalPosition;
END_IF

// Set the position prior to the move but after the reset.
mcSetPos(
    Axis:=stMotionStage.Axis,
    Execute:=bResetDone AND bExecute AND NOT bSetDone AND NOT bError,
    Position:=fStartPosition,
);
IF mcSetPos.Done OR mcSetPos.Error THEN
    nLatchError := mcSetPos.ErrorID;
END_IF
bSetDone S= mcSetPos.Done AND NOT mcSetPos.Error AND stMotionStage.stAxisStatus.fActPosition = fStartPosition;

// Any sub-error is an error here
bError := fbMoveRequest.bError OR mcSetPos.Error;

// Reset bBusy when appropriate
bBusy R= (bMoveDone AND NOT bStoppingMotor) OR bError OR ftExec.Q;

// Extract the motor position
fActPosition := stMotionStage.stAxisStatus.fActPosition;

END_FUNCTION_BLOCK

// Tests/FB_TestHelperSetAndMove_Test
FUNCTION_BLOCK FB_TestHelperSetAndMove_Test EXTENDS TcUnit.FB_TestSuite
(*
    Ensure that the test helper function block works as needed.
    Without this, all tests that need motion cannot pass.
*)
VAR
    stMotionStage: ST_MotionStage;
    fbMotionStage: FB_MotionStage;
    fbTestMove: FB_TestHelperSetAndMove;
    rtResetDone: R_TRIG;
    rtSetDone: R_TRIG;
    rtMotionStart: R_TRIG;
    rtMoveDone: R_TRIG;
END_VAR


fbMotionStage(stMotionStage:=stMotionstage);
BasicMotion();

METHOD PRIVATE BasicMotion
VAR_INPUT
END_VAR

TEST('BasicMotion');

IF NOT fbTestMove.bExecute THEN
    stMotionStage.bError := TRUE;
END_IF
fbTestMove(
    stMotionStage:=stMotionStage,
    bExecute:=TRUE,
    fStartPosition:=15.0,
    fGoalPosition:=17.0,
    fVelocity:=1.0,
    bHWEnable:=TRUE,
);
rtResetDone(CLK:=fbTestMove.bResetDone);
rtSetDone(CLK:=fbTestMove.bSetDone);
rtMotionStart(CLK:=fbTestMove.bMotionStarted);
rtMoveDone(CLK:=fbTestMove.bMoveDone);
IF rtResetDone.Q THEN
    AssertFalse(
        Condition:=stMotionStage.bError,
        Message:='Reset did not clear error',
    );
    AssertEquals_LREAL(
        Expected:=stMotionStage.stAxisStatus.fActPosition,
        Actual:=fbTestMove.fActPosition,
        Delta:=0,
        Message:='Real position output does not match real position.',
    );
END_IF
IF rtSetDone.Q THEN
    AssertEquals_LREAL(
        Expected:=fbTestMove.fStartPosition,
        Actual:=fbTestMove.fActPosition,
        Delta:=0,
        Message:='Was not set to start position after set done',
    );
END_IF
IF rtMotionStart.Q THEN
    AssertTrue(
        Condition:=stMotionStage.bBusy,
        Message:='stMotionStage is not busy, but motion is said to have started.',
    );
    AssertTrue(
        Condition:=fbTestMove.fActPosition > fbTestMove.fStartPosition,
        Message:='stMotionStage has not moved, but motion is said to have started.',
    );
END_IF
IF rtMoveDone.Q THEN
    AssertEquals_LREAL(
        Expected:=fbTestMove.fGoalPosition,
        Actual:=fbTestMove.fActPosition,
        Delta:=0.001,
        Message:='Did not reach destination at move done',
    );
END_IF
IF fbTestMove.bError OR fbTestMove.tElapsed > T#5s OR (fbTestMove.bResetDone AND fbTestMove.bSetDone AND fbTestMove.bMotionStarted AND fbTestMove.bMoveDone) THEN
    AssertFalse(
        Condition:=fbTestMove.bError,
        Message:='Error in fbTestMove',
    );
    AssertFalse(
        Condition:=fbTestMove.tElapsed > T#5s,
        Message:='Timeout in basic motion test',
    );
    TEST_FINISHED();
END_IF
END_METHOD

END_FUNCTION_BLOCK

// Tests/FB_AtPositionState_Test
FUNCTION_BLOCK FB_AtPositionState_Test EXTENDS TcUnit.FB_TestSuite
(*
    Test the following related helper functions:
    - F_PosOverLowerBound
    - F_PosUnderUpperBound
    - F_PosWithinDelta
    - F_AtPositionState
*)
VAR
    // For the multi-cycle tests
    stMotionStage: ST_MotionStage;
    fbMotionStage: FB_MotionStage;
    fbTestMove: FB_TestHelperSetAndMove;
    stPositionStateInactive: ST_PositionState;
    stPositionStateInvalid: ST_PositionState;
    stPositionStateGood: ST_PositionState;
    tonInactive: TON;
    fbInternalGood: FB_PositionStateInternal;
    fbInternalInvalid: FB_PositionStateInternal;
    nTestCounter: UINT;
    bOneTestDone: BOOL;
END_VAR


// Single cycle tests
TestPosOverLowerBoundYes();
TestPosOverLowerBoundNo();
TestPosUnderUpperBoundYes();
TestPosUnderUpperBoundNo();
TestPosWithinDeltaTooLow();
TestPosWithinDeltaTooHigh();
TestPosWithinDeltaJustRight();

// Multi cycle tests
fbMotionStage(stMotionStage:=stMotionStage);
stPositionStateInactive.sName := 'Inactive';
stPositionStateInactive.fPosition := 30.0;
stPositionStateInactive.fDelta := 1.0;
stPositionStateInactive.bValid := TRUE;
tonInactive(
    IN:=TRUE,
    PT:=T#1s,
);
TestAtPositionStateWithoutInternal();

stPositionStateInvalid.sName := 'Invalid';
stPositionStateInvalid.fPosition := 40.0;
stPositionStateInvalid.fDelta := 1.0;
stPositionStateInvalid.bValid := FALSE;
fbInternalInvalid(
    stMotionStage:=stMotionStage,
    stPositionState:=stPositionStateInvalid,
);
TestAtPositionStateInvalid();

stPositionStateGood.sName := 'Good';
stPositionStateGood.fPosition := 50.0;
stPositionStateGood.fDelta := 1.0;
stPositionStateGood.bValid := TRUE;
fbInternalGood(
    stMotionStage:=stMotionStage,
    stPositionState:=stPositionStateGood,
);
TestAtPositionStateTooLow();
TestAtPositionStateTooHigh();
TestAtPositionStateJustRight();
TestAtPositionStateTweak();
TestAtPositionStateLeave();

IF bOneTestDone THEN
    bOneTestDone := FALSE;
    nTestCounter := nTestCounter + 1;
    fbTestMove(
        stMotionStage:=stMotionStage,
        bExecute:=FALSE,
    );
END_IF

METHOD PRIVATE TestAtPositionStateInvalid
(*
    If a position state is invalid, it is never the right state.
*)
VAR

END_VAR

TEST('TestAtPositionStateInvalid');
IF nTestCounter <> 1 THEN
    RETURN;
END_IF

fbTestMove(
    stMotionStage:=stMotionstage,
    bExecute:=TRUE,
    fStartPosition:=stPositionStateInvalid.fPosition,
    fGoalPosition:=stPositionStateInvalid.fPosition,
);
IF fbTestMove.tElapsed > T#1s OR (stPositionStateInvalid.bUpdated AND fbTestMove.bSetDone) THEN
    AssertFalse(
        Condition:=F_AtPositionState(
            stMotionStage:=stMotionStage,
            stPositionState:=stPositionStateInvalid,
        ),
        Message:='Invalid state was marked OK',
    );
    AssertFalse(
        Condition:=fbTestMove.tElapsed > T#1s,
        Message:='Timeout in multi cycle test',
    );
    bOneTestDone := TRUE;
    TEST_FINISHED();
END_IF
END_METHOD

METHOD PRIVATE TestAtPositionStateJustRight
VAR
    fLocalGoal: LREAL;
END_VAR

TEST('TestAtPositionStateJustRight');
IF nTestCounter <> 4 THEN
    RETURN;
END_IF

fLocalGoal := stPositionStateGood.fPosition + 0.2*stPositionStateGood.fDelta;
fbTestMove(
    stMotionStage:=stMotionstage,
    bExecute:=TRUE,
    fStartPosition:=fLocalGoal,
    fGoalPosition:=fLocalGoal,
);
IF fbTestMove.tElapsed > T#1s OR (stPositionStateGood.bUpdated AND fbTestMove.bSetDone) THEN
    AssertTrue(
        Condition:=F_AtPositionState(
            stMotionStage:=stMotionStage,
            stPositionState:=stPositionStateGood,
        ),
        Message:='Within delta counted as outside range',
    );
    AssertFalse(
        Condition:=fbTestMove.tElapsed > T#1s,
        Message:='Timeout in multi cycle test',
    );
    bOneTestDone := TRUE;
    TEST_FINISHED();
END_IF
END_METHOD

METHOD PRIVATE TestAtPositionStateLeave
(*
    A move away from a state should be not at the state, even before we've left
*)
VAR
END_VAR

TEST('TestAtPositionStateLeave');
IF nTestCounter <> 6 THEN
    RETURN;
END_IF

fbTestMove(
    stMotionStage:=stMotionStage,
    bExecute:=TRUE,
    fStartPosition:=stPositionStateGood.fPosition,
    fGoalPosition:=stPositionStateGood.fPosition + 100 * stPositionStateGood.fDelta,
    fVelocity:=0.001,
    bHWEnable:=TRUE,
);

IF fbTestMove.tElapsed > T#5s OR (stPositionStateGood.bUpdated AND fbTestMove.bMotionStarted) THEN
    AssertTrue(
        Condition:=fbTestMove.fActPosition < stPositionStateGood.fPosition + stPositionStateGood.fDelta,
        Message:='We must be at the state location still to properly run this test.',
    );
    AssertFalse(
        Condition:=F_AtPositionState(
            stMotionStage:=stMotionStage,
            stPositionState:=stPositionStateGood,
        ),
        Message:='Leaving state is not at state once the move starts',
    );
    AssertFalse(
        Condition:=fbTestMove.tElapsed > T#5s,
        Message:='Timeout in multi cycle test',
    );
    bOneTestDone := TRUE;
    TEST_FINISHED();
END_IF
END_METHOD

METHOD PRIVATE TestAtPositionStateTooHigh
VAR
    fLocalGoal: LREAL;
END_VAR

TEST('TestAtPositionStateTooHigh');
IF nTestCounter <> 3 THEN
    RETURN;
END_IF

fLocalGoal := stPositionStateGood.fPosition + 2*stPositionStateGood.fDelta;
fbTestMove(
    stMotionStage:=stMotionstage,
    bExecute:=TRUE,
    fStartPosition:=fLocalGoal,
    fGoalPosition:=fLocalGoal,
);
IF fbTestMove.tElapsed > T#1s OR (stPositionStateGood.bUpdated AND fbTestMove.bSetDone) THEN
    AssertFalse(
        Condition:=F_AtPositionState(
            stMotionStage:=stMotionStage,
            stPositionState:=stPositionStateGood,
        ),
        Message:='Above delta counted as in range',
    );
    AssertFalse(
        Condition:=fbTestMove.tElapsed > T#1s,
        Message:='Timeout in multi cycle test',
    );
    bOneTestDone := TRUE;
    TEST_FINISHED();
END_IF
END_METHOD

METHOD PRIVATE TestAtPositionStateTooLow
VAR
    fLocalGoal: LREAL;
END_VAR

TEST('TestAtPositionStateTooLow');
IF nTestCounter <> 2 THEN
    RETURN;
END_IF

fLocalGoal := stPositionStateGood.fPosition - 2*stPositionStateGood.fDelta;
fbTestMove(
    stMotionStage:=stMotionstage,
    bExecute:=TRUE,
    fStartPosition:=fLocalGoal,
    fGoalPosition:=fLocalGoal,
);
IF fbTestMove.tElapsed > T#1s OR (stPositionStateGood.bUpdated AND fbTestMove.bSetDone) THEN
    AssertFalse(
        Condition:=F_AtPositionState(
            stMotionStage:=stMotionStage,
            stPositionState:=stPositionStateGood,
        ),
        Message:='Below delta counted as in range',
    );
    AssertFalse(
        Condition:=fbTestMove.tElapsed > T#1s,
        Message:='Timeout in multi cycle test',
    );
    bOneTestDone := TRUE;
    TEST_FINISHED();
END_IF
END_METHOD

METHOD PRIVATE TestAtPositionStateTweak
(*
    A small tweak move within the delta of a position state should be OK
*)
VAR

END_VAR

TEST('TestAtPositionStateTweak');
IF nTestCounter <> 5 THEN
    RETURN;
END_IF

fbTestMove(
    stMotionStage:=stMotionStage,
    bExecute:=TRUE,
    fStartPosition:=stPositionStateGood.fPosition,
    fGoalPosition:=stPositionStateGood.fPosition + 0.9 * stPositionStateGood.fDelta,
    fVelocity:=0.001,
    bHWEnable:=TRUE,
);

IF fbTestMove.tElapsed > T#5s OR (stPositionStateGood.bUpdated AND fbTestMove.bMotionStarted) THEN
    AssertTrue(
        Condition:=F_AtPositionState(
            stMotionStage:=stMotionStage,
            stPositionState:=stPositionStateGood,
        ),
        Message:='Small tweak in range should count as at state',
    );
    AssertFalse(
        Condition:=fbTestMove.tElapsed > T#5s,
        Message:='Timeout in multi cycle test',
    );
    bOneTestDone := TRUE;
    TEST_FINISHED();
END_IF
END_METHOD

METHOD PRIVATE TestAtPositionStateWithoutInternal
(*
    If a position state is never updated by the internal FB, it is never the right state.
*)
VAR

END_VAR

TEST('TestAtPositionStateWithoutInternal');
IF nTestCounter <> 0 THEN
    RETURN;
END_IF

fbTestMove(
    stMotionStage:=stMotionstage,
    bExecute:=TRUE,
    fStartPosition:=stPositionStateInactive.fPosition,
    fGoalPosition:=stPositionStateInactive.fPosition,
);
IF fbTestMove.tElapsed > T#1s OR (stPositionStateInvalid.bUpdated AND fbTestMove.bSetDone) THEN
    // Check for a different state to be bUpdated for timing purposes, this one never gets bUpdated
    AssertFalse(
        Condition:=F_AtPositionState(
            stMotionStage:=stMotionStage,
            stPositionState:=stPositionStateInactive,
        ),
        Message:='This is the control group, internal was not run so this should not work',
    );
    AssertFalse(
        Condition:=fbTestMove.tElapsed > T#1s,
        Message:='Timeout in multi cycle test',
    );
    bOneTestDone := TRUE;
    TEST_FINISHED();
END_IF
END_METHOD

METHOD PRIVATE TestPosOverLowerBoundNo
VAR
    stPositionState: ST_PositionState;
END_VAR

TEST('TestPosOverLowerBoundNo');
stPositionState.fPosition := 10;
stPositionState.fDelta := 1;

AssertFalse(
    Condition:=F_PosOverLowerBound(
        fPosition:=8.5,
        stPositionState:=stPositionState,
    ),
    Message:='Decided 8.5 > 9.0',
);
TEST_FINISHED();
END_METHOD

METHOD PRIVATE TestPosOverLowerBoundYes
VAR
    stPositionState: ST_PositionState;
END_VAR

TEST('TestPosOverLowerBoundYes');
stPositionState.fPosition := 10;
stPositionState.fDelta := 1;

AssertTrue(
    Condition:=F_PosOverLowerBound(
        fPosition:=9.1,
        stPositionState:=stPositionState,
    ),
    Message:='Decided 9.0 > 9.1',
);
TEST_FINISHED();
END_METHOD

METHOD PRIVATE TestPosUnderUpperBoundNo
VAR
    stPositionState: ST_PositionState;
END_VAR

TEST('TestPosUnderUpperBoundNo');
stPositionState.fPosition := 10;
stPositionState.fDelta := 1;

AssertFalse(
    Condition:=F_PosUnderUpperBound(
        fPosition:=12.0,
        stPositionState:=stPositionState,
    ),
    Message:='Decided 11.0 > 12.0',
);
TEST_FINISHED();
END_METHOD

METHOD PRIVATE TestPosUnderUpperBoundYes
VAR
    stPositionState: ST_PositionState;
END_VAR

TEST('TestPosUnderUpperBoundYes');
stPositionState.fPosition := 10;
stPositionState.fDelta := 1;

AssertTrue(
    Condition:=F_PosUnderUpperBound(
        fPosition:=10.9,
        stPositionState:=stPositionState,
    ),
    Message:='Decided 10.9 > 11.0',
);
TEST_FINISHED();
END_METHOD

METHOD PRIVATE TestPosWithinDeltaJustRight
VAR
    stPositionState: ST_PositionState;
END_VAR

TEST('TestPosWithinDeltaJustRight');
stPositionState.fPosition := 20;
stPositionState.fDelta := 1;

AssertTrue(
    Condition:=F_PosWithinDelta(
        fPosition:=20.2,
        stPositionState:=stPositionState,
    ),
    Message:='Decided 20.2 not within 19 to 21 bounds',
);
TEST_FINISHED();
END_METHOD

METHOD PRIVATE TestPosWithinDeltaTooHigh
VAR
    stPositionState: ST_PositionState;
END_VAR

TEST('TestPosWithinDeltaTooHigh');
stPositionState.fPosition := 20;
stPositionState.fDelta := 1;

AssertFalse(
    Condition:=F_PosWithinDelta(
        fPosition:=25.0,
        stPositionState:=stPositionState,
    ),
    Message:='Decided 21.0 > 25.0',
);
TEST_FINISHED();
END_METHOD

METHOD PRIVATE TestPosWithinDeltaTooLow
VAR
    stPositionState: ST_PositionState;
END_VAR

TEST('TestPosWithinDeltaTooLow');
stPositionState.fPosition := 20;
stPositionState.fDelta := 1;

AssertFalse(
    Condition:=F_PosWithinDelta(
        fPosition:=12.0,
        stPositionState:=stPositionState,
    ),
    Message:='Decided 12.0 > 19.0',
);
TEST_FINISHED();
END_METHOD

END_FUNCTION_BLOCK

// Tests/FB_AxisParameterSetExposed_Test
FUNCTION_BLOCK FB_AxisParameterSetExposed_Test EXTENDS FB_MotorTestSuite
(*
    Quick Check to verify exposed NC parameters are copied properly.
*)
VAR
    stMotionStage: ST_MotionStage;
    fbMotionStage: FB_MotionStage;
    nTestCounter: UINT;
    bOneTestDone: BOOL;
    tonTimer: TON;
END_VAR

IF nTestCounter = 0 THEN
    nTestCounter := 1;
END_IF

// Test that parameters are copied to the exposed parameters properly.
TestParameterCopy(1);

IF bOneTestDone THEN
    bOneTestDone := FALSE;
    nTestCounter := nTestCounter + 1;
    tonTimer(IN:=FALSE);
END_IF;

// Use this timer to time out any tests that stall
tonTimer(
    IN:=nTestCounter >= 1,
    PT:=T#2s,
);

METHOD TestParameterCopy
VAR_INPUT
    nTestIndex: UINT;
END_VAR
VAR_INST
    bLocalInit: BOOL := TRUE;
    bAllModified: BOOL;
    bReady: BOOL;
    bDone: BOOL;
END_VAR
TEST(CONCAT('TestParameterCopy', UINT_TO_STRING(nTestIndex)));
IF nTestCounter <> nTestIndex OR bOneTestDone THEN
    RETURN;
END_IF

fbMotionStage(stMotionStage:=stMotionStage);

IF bLocalInit THEN
    stMotionStage.stAxisParametersExposed.bCtrlEnablePosDiffControl     := 100;
    stMotionStage.stAxisParametersExposed.bEncEnableSoftEndMaxControl   := 101;
    stMotionStage.stAxisParametersExposed.bEncEnableSoftEndMinControl   := 102;
    stMotionStage.stAxisParametersExposed.fAccelerationMax              := 103;
    stMotionStage.stAxisParametersExposed.fCtrlPosDiffMax               := 104;
    stMotionStage.stAxisParametersExposed.fCtrlPosDiffMaxTime           := 105;
    stMotionStage.stAxisParametersExposed.fDecelerationMax              := 106;
    stMotionStage.stAxisParametersExposed.fEncSoftEndMax                := 107;
    stMotionStage.stAxisParametersExposed.fEncSoftEndMin                := 108;
    stMotionStage.stAxisParametersExposed.fVeloMaximum                  := 109;
    stMotionStage.stAxisParametersExposed.fEncOffset					:= 110;
    stMotionStage.stAxisParametersExposed.fEncScaleFactorInternal		:= 111;

    bLocalInit := FALSE;

    bAllModified :=
        stMotionStage.stAxisParametersExposed.bCtrlEnablePosDiffControl     <> stMotionStage.stAxisParameters.bCtrlEnablePosDiffControl AND
        stMotionStage.stAxisParametersExposed.bEncEnableSoftEndMaxControl   <> stMotionStage.stAxisParameters.bEncEnableSoftEndMaxControl AND
        stMotionStage.stAxisParametersExposed.bEncEnableSoftEndMinControl   <> stMotionStage.stAxisParameters.bEncEnableSoftEndMinControl AND
        stMotionStage.stAxisParametersExposed.fAccelerationMax              <> stMotionStage.stAxisParameters.fAccelerationMax AND
        stMotionStage.stAxisParametersExposed.fCtrlPosDiffMax               <> stMotionStage.stAxisParameters.fCtrlPosDiffMax AND
        stMotionStage.stAxisParametersExposed.fCtrlPosDiffMaxTime           <> stMotionStage.stAxisParameters.fCtrlPosDiffMaxTime AND
        stMotionStage.stAxisParametersExposed.fDecelerationMax              <> stMotionStage.stAxisParameters.fDecelerationMax AND
        stMotionStage.stAxisParametersExposed.fEncSoftEndMax                <> stMotionStage.stAxisParameters.fEncSoftEndMax AND
        stMotionStage.stAxisParametersExposed.fEncSoftEndMin                <> stMotionStage.stAxisParameters.fEncSoftEndMin AND
        stMotionStage.stAxisParametersExposed.fVeloMaximum                  <> stMotionStage.stAxisParameters.fVeloMaximum AND
        stMotionStage.stAxisParametersExposed.fEncOffset                	<> stMotionStage.stAxisParameters.fEncOffset AND
        stMotionStage.stAxisParametersExposed.fEncScaleFactorInternal       <> stMotionStage.stAxisParameters.fEncScaleFactorInternal;

    AssertTrue(
        Condition:=bAllModified,
        Message:='One or more parameters was not modified initially so the check is invalid.',
    );
END_IF

bReady :=
        stMotionStage.stAxisParameters.bCtrlEnablePosDiffControl     <> 0 AND
        stMotionStage.stAxisParameters.bEncEnableSoftEndMaxControl   <> 0 AND
        stMotionStage.stAxisParameters.bEncEnableSoftEndMinControl   <> 0 AND
        stMotionStage.stAxisParameters.fAccelerationMax              <> 0 AND
        stMotionStage.stAxisParameters.fCtrlPosDiffMax               <> 0 AND
        stMotionStage.stAxisParameters.fCtrlPosDiffMaxTime           <> 0 AND
        stMotionStage.stAxisParameters.fDecelerationMax              <> 0 AND
        stMotionStage.stAxisParameters.fEncSoftEndMax                <> 0 AND
        stMotionStage.stAxisParameters.fEncSoftEndMin                <> 0 AND
        stMotionStage.stAxisParameters.fVeloMaximum                  <> 0 AND
        stMotionStage.stAxisParameters.fEncOffset					 <> 0 AND
        stMotionStage.stAxisParameters.fEncScaleFactorInternal       <> 0;

IF bReady THEN
    bDone :=
        stMotionStage.stAxisParametersExposed.bCtrlEnablePosDiffControl     = stMotionStage.stAxisParameters.bCtrlEnablePosDiffControl AND
        stMotionStage.stAxisParametersExposed.bEncEnableSoftEndMaxControl   = stMotionStage.stAxisParameters.bEncEnableSoftEndMaxControl AND
        stMotionStage.stAxisParametersExposed.bEncEnableSoftEndMinControl   = stMotionStage.stAxisParameters.bEncEnableSoftEndMinControl AND
        stMotionStage.stAxisParametersExposed.fAccelerationMax              = stMotionStage.stAxisParameters.fAccelerationMax AND
        stMotionStage.stAxisParametersExposed.fCtrlPosDiffMax               = stMotionStage.stAxisParameters.fCtrlPosDiffMax AND
        stMotionStage.stAxisParametersExposed.fCtrlPosDiffMaxTime           = stMotionStage.stAxisParameters.fCtrlPosDiffMaxTime AND
        stMotionStage.stAxisParametersExposed.fDecelerationMax              = stMotionStage.stAxisParameters.fDecelerationMax AND
        stMotionStage.stAxisParametersExposed.fEncSoftEndMax                = stMotionStage.stAxisParameters.fEncSoftEndMax AND
        stMotionStage.stAxisParametersExposed.fEncSoftEndMin                = stMotionStage.stAxisParameters.fEncSoftEndMin AND
        stMotionStage.stAxisParametersExposed.fVeloMaximum                  = stMotionStage.stAxisParameters.fVeloMaximum AND
        stMotionStage.stAxisParametersExposed.fEncOffset                	= stMotionStage.stAxisParameters.fEncOffset AND
        stMotionStage.stAxisParametersExposed.fEncScaleFactorInternal       = stMotionStage.stAxisParameters.fEncScaleFactorInternal;
END_IF

IF bDone OR tonTimer.Q THEN
    AssertFalse(
        Condition:=tonTimer.Q,
        Message:=CONCAT(CONCAT('Failed to update the parameters within ', TIME_TO_STRING(tonTimer.PT)),' seconds.'),
    );
    AssertTrue(
        Condition:=bDone,
        Message:='One or more parameters was not copied properly.',
    );

    bOneTestDone := TRUE;
    TEST_FINISHED();
END_IF
END_METHOD

END_FUNCTION_BLOCK

// Tests/FB_MiscStatesErrorFFO_Test
FUNCTION_BLOCK FB_MiscStatesErrorFFO_Test EXTENDS TcUnit.FB_TestSuite
(*
    Unit tests for FB_MiscStatesErrorFFO
*)
VAR
END_VAR


TestBeamParamsNotOk();
TestZeroRate();
TestUnknownState();
TestTransitionState();
TestDebounce();

METHOD TestBeamParamsNotOk
VAR_INST
    fbMiscFFO: FB_MiscStatesErrorFFO;
    fbArbiter: FB_Arbiter(1);
    fbFFHWO: FB_HardwareFFOutput := (bAutoReset := TRUE);

    stBeamReq: ST_BeamParams;
END_VAR

TEST('TestBeamParamsNotOk');

fbFFHWO.EvaluateOutput();
AssertTrue(
    fbFFHWO.q_xFastFaultOut,
    'Started with a fault',
);

// Trigger only a beam parameter mismatch
// Do not trip zero rate, unknown state, or debounce
PMPS_GVL.stCurrentBeamParameters := PMPS_GVL.cstFullBeam;
stBeamReq := PMPS_GVL.cstFullBeam;
stBeamReq.nTran := 0.5;
fbMiscFFO(
    fbArbiter:=fbArbiter,
    fbFFHWO:=fbFFHWO,
    stCurrentBeamReq:=stBeamReq,
    bKnownState:=TRUE,
    nTransitionID:=1,
);

fbFFHWO.EvaluateOutput();
AssertFalse(
    fbFFHWO.q_xFastFaultOut,
    'Did not fault with bad attenuator state',
);

TEST_FINISHED();
END_METHOD

METHOD TestDebounce
VAR_INST
    fbMiscFFO: FB_MiscStatesErrorFFO;
    fbArbiter: FB_Arbiter(5);
    fbFFHWO: FB_HardwareFFOutput := (bAutoReset := TRUE);
END_VAR
VAR
    nIter: DINT;
END_VAR

TEST('TestDebounce');

fbFFHWO.EvaluateOutput();
AssertTrue(
    fbFFHWO.q_xFastFaultOut,
    'Started with a fault prior to first FB run-through',
);
// Ask for full beam: there should be no faults of any kind
fbMiscFFO(
    fbArbiter:=fbArbiter,
    fbFFHWO:=fbFFHWO,
    stCurrentBeamReq:=PMPS_GVL.cstFullBeam,
    bKnownState:=TRUE,
    nTransitionID:=5,
);
fbFFHWO.EvaluateOutput();

AssertTrue(
    fbFFHWO.q_xFastFaultOut,
    'Started with a fault prior to trip checks',
);

// Trip and untrip the beam fast fault once, show no fault
TripUntrip(
    fbMiscFFO:=fbMiscFFO,
    fbArbiter:=fbArbiter,
    fbFFHWO:=fbFFHWO,
);
AssertTrue(
    fbFFHWO.q_xFastFaultOut,
    'Control group failed: one trip/untrip should not be enough to debounce',
);
// Trip and untrip the beam fast fault like 10 times, show fault
FOR nIter := 1 TO 10 DO
    TripUntrip(
        fbMiscFFO:=fbMiscFFO,
        fbArbiter:=fbArbiter,
        fbFFHWO:=fbFFHWO,
    );
END_FOR
AssertFalse(
    fbFFHWO.q_xFastFaultOut,
    'Debouncer failed to debounce',
);

TEST_FINISHED();
END_METHOD

METHOD TestTransitionState
VAR_INST
    fbMiscFFO: FB_MiscStatesErrorFFO;
    fbArbiter: FB_Arbiter(4);
    fbFFHWO: FB_HardwareFFOutput := (bAutoReset := TRUE);
END_VAR

TEST('TestTransitionState');

fbFFHWO.EvaluateOutput();
AssertTrue(
    fbFFHWO.q_xFastFaultOut,
    'Started with a fault',
);

// Trigger no faults, we're at an unknown state but it's a transition state
// Do not trip bad beam, zero rate, or debounce
fbArbiter.AddRequest(
    nReqID:=4,
    stReqBP:=PMPS_GVL.cstFullBeam,
    sDevName:='UnitTest',
);
PMPS_GVL.stCurrentBeamParameters := PMPS_GVL.cstFullBeam;
fbMiscFFO(
    fbArbiter:=fbArbiter,
    fbFFHWO:=fbFFHWO,
    stCurrentBeamReq:=PMPS_GVL.cstFullBeam,
    bKnownState:=FALSE,
    nTransitionID:=4,
);

fbFFHWO.EvaluateOutput();
AssertTrue(
    fbFFHWO.q_xFastFaultOut,
    'Faulted in unknown states even though we were moving normally',
);

TEST_FINISHED();
END_METHOD

METHOD TestUnknownState
VAR_INST
    fbMiscFFO: FB_MiscStatesErrorFFO;
    fbArbiter: FB_Arbiter(3);
    fbFFHWO: FB_HardwareFFOutput := (bAutoReset := TRUE);
END_VAR

TEST('TestUnknownState');

fbFFHWO.EvaluateOutput();
AssertTrue(
    fbFFHWO.q_xFastFaultOut,
    'Started with a fault',
);

// Trigger only an unknown states
// Do not trip bad beam, zero rate, or debounce
PMPS_GVL.stCurrentBeamParameters := PMPS_GVL.cstFullBeam;
fbMiscFFO(
    fbArbiter:=fbArbiter,
    fbFFHWO:=fbFFHWO,
    stCurrentBeamReq:=PMPS_GVL.cstFullBeam,
    bKnownState:=FALSE,
    nTransitionID:=3,
);

fbFFHWO.EvaluateOutput();
AssertFalse(
    fbFFHWO.q_xFastFaultOut,
    'Did not fault with unknown state',
);

TEST_FINISHED();
END_METHOD

METHOD TestZeroRate
VAR_INST
    fbMiscFFO: FB_MiscStatesErrorFFO;
    fbArbiter: FB_Arbiter(2);
    fbFFHWO: FB_HardwareFFOutput := (bAutoReset := TRUE);

    stNoBeam: ST_BeamParams;
END_VAR

TEST('TestBeamZeroRate');

fbFFHWO.EvaluateOutput();
AssertTrue(
    fbFFHWO.q_xFastFaultOut,
    'Started with a fault',
);

// Trigger only a zero rate
// Do not trip beam parameter mismatch, unknown state, or debounce
PMPS_GVL.stCurrentBeamParameters := stNoBeam;
fbMiscFFO(
    fbArbiter:=fbArbiter,
    fbFFHWO:=fbFFHWO,
    stCurrentBeamReq:=PMPS_GVL.cst0RateBeam,
    bKnownState:=TRUE,
    nTransitionID:=2
);

fbFFHWO.EvaluateOutput();
AssertFalse(
    fbFFHWO.q_xFastFaultOut,
    'Did not fault with zero rate',
);

TEST_FINISHED();
END_METHOD

METHOD TripUntrip
VAR_IN_OUT
    fbMiscFFO: FB_MiscStatesErrorFFO;
    fbArbiter: FB_Arbiter;
    fbFFHWO: FB_HardwareFFOutput;
END_VAR
VAR
    stBeamReq: ST_BeamParams;
END_VAR

// Use anything other than 0 rate, which is its own check
stBeamReq := PMPS_GVL.cstFullBeam;
stBeamReq.nTran := 0.5;
// Trip: too much beam!
PMPS_GVL.stCurrentBeamParameters := PMPS_GVL.cstFullBeam;
fbMiscFFO(
    fbArbiter:=fbArbiter,
    fbFFHWO:=fbFFHWO,
    stCurrentBeamReq:=stBeamReq,
    bKnownState:=TRUE,
    nTransitionID:=5,
);
fbFFHWO.EvaluateOutput();

// Untrip: correct beam!
PMPS_GVL.stCurrentBeamParameters := stBeamReq;
fbMiscFFO(
    fbArbiter:=fbArbiter,
    fbFFHWO:=fbFFHWO,
    stCurrentBeamReq:=stBeamReq,
    bKnownState:=TRUE,
    nTransitionID:=5,
);
fbFFHWO.EvaluateOutput();
END_METHOD

END_FUNCTION_BLOCK

// Tests/FB_MotionBPTM_Test
FUNCTION_BLOCK FB_MotionBPTM_Test EXTENDS TcUnit.FB_TestSuite
(*
    Test the functionality of the motion bptm,
    Which is just a bptm wrapped up with a set of n motors.
    We're basically just making sure that we push the done button at the appropriate time.
    Direct tests of BPTM itself are reserved for the pmps library.

    The BPTM takes care of these executions across multiple cycles,
    so these tests must implement timeouts.
*)
VAR
    astMotionStage: ARRAY[1..MotionConstants.MAX_STATE_MOTORS] OF ST_MotionStage;
    stGoal1: ST_DbStateParams;
    stGoal2: ST_DbStateParams;
    stTrans: ST_DbStateParams;
    stNoBeam: ST_BeamParams;
END_VAR


stGoal1.stBeamParams := PMPS_GVL.cstFullBeam;
stGoal1.nRequestAssertionID := 1;
stGoal1.sPmpsState := 'stGoal1';
stGoal2.stBeamParams := PMPS_GVL.cstFullBeam;
stGoal2.stBeamParams.nTran := 0.5;
stGoal2.nRequestAssertionID := 2;
stGoal2.sPmpsState := 'stGoal2';
stTrans.stBeamParams := PMPS_GVL.cst0RateBeam;
stTrans.nRequestAssertionID := 3;
stTrans.sPmpsState := 'stTrans';

// Just put a blanket global no beam so these won't wait for any changes ever
PMPS_GVL.stCurrentBeamParameters := stNoBeam;
TestInit();
Test3dMove();
TestNoMove();
TestCount();

METHOD AssertInPool
VAR_IN_OUT
    fbArbiter: FB_Arbiter;
    stDbStateParams: ST_DbStateParams;
END_VAR
VAR_INPUT
    bInPool: BOOL;
    sContext: STRING;
END_VAR

IF bInPool THEN
    AssertTrue(
        fbArbiter.CheckRequestInPool(stDbStateParams.nRequestAssertionID),
        CONCAT(CONCAT(stDbStateParams.sPmpsState, ' Beam parameters were not in the pool '), sContext),
    );
ELSE
    AssertFalse(
        fbArbiter.CheckRequestInPool(stDbStateParams.nRequestAssertionID),
        CONCAT(CONCAT(stDbStateParams.sPmpsState, ' Beam parameters unexpectedly found in the pool '), sContext),
    );
END_IF
END_METHOD

METHOD SetMotorDone
VAR_INPUT
END_VAR

// Force post-move state
astMotionStage[1].bBusy := FALSE;
astMotionStage[1].bDone := TRUE;
astMotionStage[2].bBusy := FALSE;
astMotionStage[2].bDone := TRUE;
astMotionStage[3].bBusy := FALSE;
astMotionStage[3].bDone := TRUE;
END_METHOD

METHOD SetMotorMoving
VAR_INPUT
END_VAR

// Force a moving but not done state
astMotionStage[1].bBusy := TRUE;
astMotionStage[1].bDone := FALSE;
astMotionStage[2].bBusy := TRUE;
astMotionStage[2].bDone := FALSE;
astMotionStage[3].bBusy := TRUE;
astMotionStage[3].bDone := FALSE;
END_METHOD

METHOD SetMotorStartup
VAR_INPUT
END_VAR

// Force some sort of default looking state
astMotionStage[1].bBusy := FALSE;
astMotionStage[1].bDone := FALSE;
astMotionStage[2].bBusy := FALSE;
astMotionStage[2].bDone := FALSE;
astMotionStage[3].bBusy := FALSE;
astMotionStage[3].bDone := FALSE;
END_METHOD

METHOD Test3dMove : BOOL
(*
    Can we safely do a 3d move?
*)
VAR_INST
    fbBptm: FB_MotionBPTM;
    fbArbiter: FB_Arbiter(2);
    fbFFHWO: FB_HardwareFFOutput := (bAutoReset := TRUE);
    fbSubSysIO : FB_DummyArbIO;

    nState: UINT;
    tonTimer: TON;
END_VAR

TEST('Test3DMove');

tonTimer(
    IN:=TRUE,
    PT:=T#5s,
);
IF tonTimer.Q THEN
    nState := 4;
END_IF

CASE nState OF
    0:
        // Establish baseline at Goal1
        SetMotorStartup();
        fbBptm(
            astMotionStage:=astMotionStage,
            fbArbiter:=fbArbiter,
            fbFFHWO:=fbFFHWO,
            stGoalParams:=stGoal1,
            stTransParams:=stTrans,
            nActiveMotorCount:=3,
            bEnable:=TRUE,
            bAtState:=TRUE,
        );
        IF fbBptm.bDone THEN
            nState := 1;
        END_IF
    1:
        // Request a move
        SetMotorStartup();
        fbBptm(
            astMotionStage:=astMotionStage,
            fbArbiter:=fbArbiter,
            fbFFHWO:=fbFFHWO,
            stGoalParams:=stGoal2,
            stTransParams:=stTrans,
            nActiveMotorCount:=3,
            bEnable:=TRUE,
            bAtState:=FALSE,
        );
        IF fbBptm.bTransitionAuthorized THEN
            // We should have transition and goal 2 asserts in
            AssertInPool(fbArbiter, stGoal1, FALSE, 'with trans auth');
            AssertInPool(fbArbiter, stGoal2, TRUE, 'with trans auth');
            AssertInPool(fbArbiter, stTrans, TRUE, 'with trans auth');
            nState := 2;
        END_IF
    2:
        // Simulate a move
        SetMotorMoving();
        fbBptm(
            astMotionStage:=astMotionStage,
            fbArbiter:=fbArbiter,
            fbFFHWO:=fbFFHWO,
            stGoalParams:=stGoal2,
            stTransParams:=stTrans,
            nActiveMotorCount:=3,
            bEnable:=TRUE,
            bAtState:=FALSE,
        );
        // Same situation as before
        AssertInPool(fbArbiter, stGoal1, FALSE, 'after move started');
        AssertInPool(fbArbiter, stGoal2, TRUE, 'after move started');
        AssertInPool(fbArbiter, stTrans, TRUE, 'after move started');
        nState := 3;
    3:
        // Move is done
        SetMotorDone();
        fbBptm(
            astMotionStage:=astMotionStage,
            fbArbiter:=fbArbiter,
            fbFFHWO:=fbFFHWO,
            stGoalParams:=stGoal2,
            stTransParams:=stTrans,
            nActiveMotorCount:=3,
            bEnable:=TRUE,
            bAtState:=TRUE,
        );
        IF fbBptm.bDone THEN
            // Dropped the transition assert
            AssertInPool(fbArbiter, stGoal1, FALSE, 'with move complete');
            AssertInPool(fbArbiter, stGoal2, TRUE, 'with move complete');
            AssertInPool(fbArbiter, stTrans, FALSE, 'with move complete');
            nState := 4;
        END_IF
    4:
        AssertFalse(
            tonTimer.Q,
            'Timeout in test',
        );
        TEST_FINISHED();
END_CASE

fbSubSysIO(
    LA:=fbArbiter,
    FFO:=fbFFHWO,
);
END_METHOD

METHOD TestCount
(*
    FB Should just error out if we forgot to give a count
*)
VAR_INST
    fbBptm: FB_MotionBPTM;
    fbArbiter: FB_Arbiter(1);
    fbFFHWO: FB_HardwareFFOutput := (bAutoReset := TRUE);

    tonWait: TON;
END_VAR
TEST('TestCount');

SetMotorStartup();
fbBptm(
    astMotionStage:=astMotionStage,
    fbArbiter:=fbArbiter,
    fbFFHWO:=fbFFHWO,
    stGoalParams:=stGoal1,
    stTransParams:=stTrans,
    bEnable:=True,
    bAtState:=True,
);
AssertTrue(
    fbBptm.bMotorCountError,
    'Did not properly error on missing motor count',
);

tonWait(
    IN:=TRUE,
    PT:=T#1s,
);
IF tonWait.Q THEN
    // Should have no arbiter activity at all
    AssertInPool(fbArbiter, stGoal1, FALSE, 'with bad count');
    AssertInPool(fbArbiter, stGoal2, FALSE, 'with bad count');
    AssertInPool(fbArbiter, stTrans, FALSE, 'with bad count');

    TEST_FINISHED();
END_IF
END_METHOD

METHOD TestInit : BOOL
(*
    If we initialize with still motors, do we get an arbiter request at the current goal? Hopefully we do.
*)
VAR_INST
    fbBptm: FB_MotionBPTM;
    fbArbiter: FB_Arbiter(1);
    fbFFHWO: FB_HardwareFFOutput := (bAutoReset := TRUE);
    fbSubSysIO : FB_DummyArbIO;

    tonTimer: TON;
END_VAR

TEST('TestInit');

SetMotorStartup();
fbBptm(
    astMotionStage:=astMotionStage,
    fbArbiter:=fbArbiter,
    fbFFHWO:=fbFFHWO,
    stGoalParams:=stGoal1,
    stTransParams:=stTrans,
    nActiveMotorCount:=3,
    bEnable:=True,
    bAtState:=True,
);
fbSubSysIO(
    LA:=fbArbiter,
    FFO:=fbFFHWO,
);

tonTimer(
    IN:=TRUE,
    PT:=T#5s,
);
IF tonTimer.Q OR fbBptm.bDone THEN
    AssertFalse(
        tonTimer.Q,
        'Timeout in test',
    );
    // We should have a request in the pool for goal 1 but not for transition
    // If no request are in the pool, we may come up in a no protection state!
    // If both requests are in the pool, we may come up in a too much blocking beam state!
    AssertInPool(fbArbiter, stGoal1, TRUE, 'at startup');
    AssertInPool(fbArbiter, stTrans, FALSE, 'at startup');

    TEST_FINISHED();
END_IF
END_METHOD

METHOD TestNoMove
(*
    In place transitions should work at startup and also at done positions.
*)
VAR_INST
    fbBptm: FB_MotionBPTM;
    fbArbiter: FB_Arbiter(1);
    fbFFHWO: FB_HardwareFFOutput := (bAutoReset := TRUE);
    fbSubSysIO : FB_DummyArbIO;

    nState: UINT;
    tonTimer: TON;
END_VAR

TEST('TestNoMove');

tonTimer(
    IN:=TRUE,
    PT:=T#5s,
);
IF tonTimer.Q THEN
    nState := 3;
END_IF

CASE nState OF
    0:
        SetMotorStartup();
        fbBptm(
            astMotionStage:=astMotionStage,
            fbArbiter:=fbArbiter,
            fbFFHWO:=fbFFHWO,
            stGoalParams:=stGoal1,
            stTransParams:=stTrans,
            nActiveMotorCount:=3,
            bEnable:=True,
            bAtState:=True,
        );
        IF fbBptm.bDone THEN
            nState := 1;
        END_IF
    1:
        SetMotorStartup();
        // NOTE: we kept bAtState TRUE the whole time, so this should be a completed in-place transition
        fbBptm(
            astMotionStage:=astMotionStage,
            fbArbiter:=fbArbiter,
            fbFFHWO:=fbFFHWO,
            stGoalParams:=stGoal2,
            stTransParams:=stTrans,
            nActiveMotorCount:=3,
            bEnable:=True,
            bAtState:=True,
        );
        IF fbBptm.bDone THEN
            // Only Goal2 should be in the pool
            AssertInPool(fbArbiter, stGoal1, FALSE, 'after switching goals (1)');
            AssertInPool(fbArbiter, stGoal2, TRUE, 'after switching goals (1)');
            AssertInPool(fbArbiter, stTrans, FALSE, 'after switching goals (1)');
            nState := 2;
        END_IF
    2:
        // Repeat from a done position!
        SetMotorDone();
        fbBptm(
            astMotionStage:=astMotionStage,
            fbArbiter:=fbArbiter,
            fbFFHWO:=fbFFHWO,
            stGoalParams:=stGoal1,
            stTransParams:=stTrans,
            nActiveMotorCount:=3,
            bEnable:=True,
            bAtState:=True,
        );
        IF fbBptm.bDone THEN
            // Only Goal1 should be in the pool
            AssertInPool(fbArbiter, stGoal1, TRUE, 'after switching goals (2)');
            AssertInPool(fbArbiter, stGoal2, FALSE, 'after switching goals (2)');
            AssertInPool(fbArbiter, stTrans, FALSE, 'after switching goals (2)');
            nState := 3;
        END_IF
    3:
        AssertFalse(
            tonTimer.Q,
            'Timeout in test',
        );
        TEST_FINISHED();
END_CASE

fbSubSysIO(
    LA:=fbArbiter,
    FFO:=fbFFHWO,
);
END_METHOD

END_FUNCTION_BLOCK

// Tests/FB_MotionClearAsserts_Test
FUNCTION_BLOCK FB_MotionClearAsserts_Test EXTENDS TcUnit.FB_TestSuite
VAR
END_VAR


TestBasic();

METHOD TestBasic
VAR
    nIter: UINT;
END_VAR
VAR_INST
    fbClear: FB_MotionClearAsserts;
    astDbStateParams: ARRAY[0..GeneralConstants.MAX_STATES] OF ST_DbStateParams;
    fbArbiter: FB_Arbiter(1);
END_VAR

TEST('TestBasic');

FOR nIter := 0 TO GeneralConstants.MAX_STATES DO
    astDbStateParams[nIter].nRequestAssertionID := 100 + nIter;
    fbArbiter.AddRequest(
        nReqID:=100 + nIter,
        stReqBP:=PMPS_GVL.cstFullBeam,
        sDevName:='UnitTest',
    );
END_FOR

FOR nIter := 0 TO GeneralConstants.MAX_STATES DO
    AssertTrue(
        fbArbiter.CheckRequestInPool(100 + nIter),
        CONCAT(CONCAT('State ', UDINT_TO_STRING(nIter)), ' was not in the pool'),
    );
END_FOR

fbClear(
    astDbStateParams:=astDbStateParams,
    fbArbiter:=fbArbiter,
    bExecute:=TRUE,
);

FOR nIter := 0 TO GeneralConstants.MAX_STATES DO
    AssertFalse(
        fbArbiter.CheckRequestInPool(100 + nIter),
        CONCAT(CONCAT('State ', UDINT_TO_STRING(nIter)), ' was not cleared from the pool'),
    );
END_FOR

TEST_FINISHED();
END_METHOD

END_FUNCTION_BLOCK

// Tests/FB_MotionReadPMPSDBND_Test
FUNCTION_BLOCK FB_MotionReadPMPSDBND_Test EXTENDS TcUnit.FB_TestSuite
(*
    We test the actual db read in the pmps lib
    Here, we test that the correct keys are ready for the read based on the inputs.

    The user submits a transition key and all of their ST_PositionState instances from all of their motors.
    Any subset of these instances can have lookup keys.

    If only one state at the index has a lookup key, use that key.
    If more than one state at the index has the same lookup key, use that key.
    If states at the same index have different keys, that's an error and a fast fault.
    If states at different indices have the same keys, that's an error and a fast fault.
*)
VAR
    astCorrectStates: ARRAY[1..GeneralConstants.MAX_STATES] OF ST_PositionState;
    astNonsenseStates: ARRAY[1..GeneralConstants.MAX_STATES] OF ST_PositionState;
    astDuplicatedStates: ARRAY[1..GeneralConstants.MAX_STATES] OF ST_PositionState;
    astHalfFullStates: ARRAY[1..GeneralConstants.MAX_STATES] OF ST_PositionState;
    nIter: UINT;
END_VAR


// Set up the state arrays that can be used in test methods
FOR nIter := 1 TO GeneralConstants.MAX_STATES DO
    astCorrectStates[nIter].stPMPS.sPmpsState := CONCAT('State', UINT_TO_STRING(nIter));
    astNonsenseStates[nIter].stPMPS.sPmpsState := CONCAT('asdf', UINT_TO_STRING(nIter));
    IF UINT_TO_BOOL(nIter MOD 2) THEN
        astDuplicatedStates[nIter].stPMPS.sPmpsState := 'State0';
    ELSE
        astDuplicatedStates[nIter].stPMPS.sPmpsState := 'State1';
    END_IF
    IF nIter <= GeneralConstants.MAX_STATES / 2 THEN
        astHalfFullStates[nIter].stPMPS.sPmpsState := CONCAT('State', UINT_TO_STRING(nIter));
    END_IF
END_FOR

TestSolo();
TestTrio();
TestNonsense();
TestDupe();
TestBackfill();
TestHalfFull();

METHOD TestBackfill
VAR_INST
    fbRead: FB_MotionReadPMPSDBND;
    astPositionState: ARRAY[1..MotionConstants.MAX_STATE_MOTORS] OF ARRAY[1..GeneralConstants.MAX_STATES] OF ST_PositionState;
    fbFFHWO: FB_HardwareFFOutput := (bAutoReset := TRUE);
    stDefaultBP: ST_DbStateParams;
END_VAR

TEST('TestBackfill');

astPositionState[1] := astCorrectStates;
// Pick a few parameters to drop in
astPositionState[1][3].stPMPS.stBeamParams.nRate := 999;
astPositionState[2][1].stPMPS.nRequestAssertionID := 777;
astPositionState[3][2].stPMPS.bBeamParamsLoaded := NOT stDefaultBP.bBeamParamsLoaded;
fbRead(
    astPositionState:=astPositionState,
    fbFFHWO:=fbFFHWO,
    sTransitionKey:='State0',
    sDeviceName:='TestBackfill',
);
// Everything should be cleared to the defaults: the library should let us know what params got loaded (none)
AssertEquals_UDINT(
    Expected:=stDefaultBP.stBeamParams.nRate,
    Actual:=astPositionState[1][3].stPMPS.stBeamParams.nRate,
    Message:='nRate of motor 1 state 3 not backfilled',
);
AssertEquals_UDINT(
    Expected:=stDefaultBP.nRequestAssertionID,
    Actual:=astPositionState[2][1].stPMPS.nRequestAssertionID,
    Message:='nRequestAssertionID of motor 2 state 3 not backfilled',
);
AssertEquals_BOOL(
    Expected:=stDefaultBP.bBeamParamsLoaded,
    Actual:=astPositionState[3][2].stPMPS.bBeamParamsLoaded,
    Message:='bBeamParamsLoaded of motor 3 state 2 not backfilled',
);

TEST_FINISHED();
END_METHOD

METHOD TestDupe
VAR_INST
    fbRead: FB_MotionReadPMPSDBND;
    astPositionState: ARRAY[1..MotionConstants.MAX_STATE_MOTORS] OF ARRAY[1..GeneralConstants.MAX_STATES] OF ST_PositionState;
    fbFFHWO: FB_HardwareFFOutput := (bAutoReset := TRUE);
END_VAR

TEST('TestDupe');

astPositionState[1] := astDuplicatedStates;
fbRead(
    astPositionState:=astPositionState,
    fbFFHWO:=fbFFHWO,
    sTransitionKey:='State0',
    sDeviceName:='TestTrio',
);
fbFFHWO.EvaluateOutput();

AssertTrue(
    fbRead.bError,
    'Should have had an error',
);
FOR nIter := 0 TO GeneralConstants.MAX_STATES DO
    AssertEquals_STRING(
        Expected:='',
        Actual:=fbRead.astDbStateParams[nIter].sPmpsState,
        Message:=CONCAT('Errored output should have had no state names: ', UINT_TO_STRING(nIter)),
    );
END_FOR

TEST_FINISHED();
END_METHOD

METHOD TestHalfFull
VAR_INST
    fbRead: FB_MotionReadPMPSDBND;
    astPositionState: ARRAY[1..MotionConstants.MAX_STATE_MOTORS] OF ARRAY[1..GeneralConstants.MAX_STATES] OF ST_PositionState;
    fbFFHWO: FB_HardwareFFOutput := (bAutoReset := TRUE);
END_VAR

TEST('TestHalfFull');

astPositionState[1] := astHalfFullStates;
fbRead(
    astPositionState:=astPositionState,
    fbFFHWO:=fbFFHWO,
    sTransitionKey:='State0',
    sDeviceName:='TestHalfFull',
);
fbFFHWO.EvaluateOutput();

AssertFalse(
    fbRead.bError,
    'Had an error',
);
AssertEquals_STRING(
    Expected:=fbRead.sTransitionKey,
    Actual:=fbRead.astDbStateParams[0].sPmpsState,
    Message:='Output did not have the correct transition state',
);
FOR nIter := 1 TO GeneralConstants.MAX_STATES / 2 DO
    AssertEquals_STRING(
        Expected:=astCorrectStates[nIter].stPMPS.sPmpsState,
        Actual:=fbRead.astDbStateParams[nIter].sPmpsState,
        Message:=CONCAT('Output did not have the correct position state: ', UINT_TO_STRING(nIter)),
    );
END_FOR

TEST_FINISHED();
END_METHOD

METHOD TestNonsense
VAR_INST
    fbRead: FB_MotionReadPMPSDBND;
    astPositionState: ARRAY[1..MotionConstants.MAX_STATE_MOTORS] OF ARRAY[1..GeneralConstants.MAX_STATES] OF ST_PositionState;
    fbFFHWO: FB_HardwareFFOutput := (bAutoReset := TRUE);
END_VAR

TEST('TestNonsense');

astPositionState[1] := astCorrectStates;
astPositionState[2] := astNonsenseStates;
fbRead(
    astPositionState:=astPositionState,
    fbFFHWO:=fbFFHWO,
    sTransitionKey:='State0',
    sDeviceName:='TestTrio',
);
fbFFHWO.EvaluateOutput();

AssertTrue(
    fbRead.bError,
    'Should have had an error',
);
// Only the transition state should be spared from the nonsense
AssertEquals_STRING(
    Expected:='State0',
    Actual:=fbRead.astDbStateParams[0].sPmpsState,
    Message:='Transition state should be OK',
);
FOR nIter := 1 TO GeneralConstants.MAX_STATES DO
    AssertEquals_STRING(
        Expected:='',
        Actual:=fbRead.astDbStateParams[nIter].sPmpsState,
        Message:=CONCAT('Errored output should have had no state names: ', UINT_TO_STRING(nIter)),
    );
END_FOR

TEST_FINISHED();
END_METHOD

METHOD TestSolo
VAR_INST
    fbRead: FB_MotionReadPMPSDBND;
    astPositionState: ARRAY[1..MotionConstants.MAX_STATE_MOTORS] OF ARRAY[1..GeneralConstants.MAX_STATES] OF ST_PositionState;
    fbFFHWO: FB_HardwareFFOutput := (bAutoReset := TRUE);
END_VAR

TEST('TestSolo');

astPositionState[1] := astCorrectStates;
fbRead(
    astPositionState:=astPositionState,
    fbFFHWO:=fbFFHWO,
    sTransitionKey:='State0',
    sDeviceName:='TestSolo',
);
fbFFHWO.EvaluateOutput();

AssertFalse(
    fbRead.bError,
    'Had an error',
);
AssertEquals_STRING(
    Expected:=fbRead.sTransitionKey,
    Actual:=fbRead.astDbStateParams[0].sPmpsState,
    Message:='Output did not have the correct transition state',
);
FOR nIter := 1 TO GeneralConstants.MAX_STATES DO
    AssertEquals_STRING(
        Expected:=astCorrectStates[nIter].stPMPS.sPmpsState,
        Actual:=fbRead.astDbStateParams[nIter].sPmpsState,
        Message:=CONCAT('Output did not have the correct position state: ', UINT_TO_STRING(nIter)),
    );
END_FOR

TEST_FINISHED();
END_METHOD

METHOD TestTrio
VAR_INST
    fbRead: FB_MotionReadPMPSDBND;
    astPositionState: ARRAY[1..MotionConstants.MAX_STATE_MOTORS] OF ARRAY[1..GeneralConstants.MAX_STATES] OF ST_PositionState;
    fbFFHWO: FB_HardwareFFOutput := (bAutoReset := TRUE);
END_VAR

TEST('TestTrio');

astPositionState[1] := astCorrectStates;
astPositionState[2] := astCorrectStates;
astPositionState[3] := astCorrectStates;
fbRead(
    astPositionState:=astPositionState,
    fbFFHWO:=fbFFHWO,
    sTransitionKey:='State0',
    sDeviceName:='TestTrio',
);
fbFFHWO.EvaluateOutput();

AssertFalse(
    fbRead.bError,
    'Had an error',
);
AssertEquals_STRING(
    Expected:=fbRead.sTransitionKey,
    Actual:=fbRead.astDbStateParams[0].sPmpsState,
    Message:='Output did not have the correct transition state',
);
FOR nIter := 1 TO GeneralConstants.MAX_STATES DO
    AssertEquals_STRING(
        Expected:=astCorrectStates[nIter].stPMPS.sPmpsState,
        Actual:=fbRead.astDbStateParams[nIter].sPmpsState,
        Message:=CONCAT('Output did not have the correct position state: ', UINT_TO_STRING(nIter)),
    );
END_FOR

TEST_FINISHED();
END_METHOD

END_FUNCTION_BLOCK

// Tests/FB_NCErrorFFO_Test
FUNCTION_BLOCK FB_NCErrorFFO_Test EXTENDS TcUnit.FB_TestSuite
(*
    Test the following related FBs:
    - FB_NCErrorFFO
    - FB_EncErrorFFO

    These function blocks are designed to trip the beam when there
    is an NC error reported by stMotionStage.
*)
VAR
    stMotionStage: ST_MotionStage;
    fbMotionStage: FB_MotionStage;
    fbFFHWO: FB_HardwareFFOutput := (bAutoReset := TRUE);
    fbCauseNCError: FB_CauseNCError;

    fbNCErrorFFO: FB_NCErrorFFO;
    fbEncErrorFFO: FB_EncErrorFFO;

    nTestCounter: UINT;
    bOneTestDone: BOOL;
    tonTimer: TON;
END_VAR


fbMotionStage(stMotionStage:=stMotionStage);
// Limit to drive errors so I can isolate it from the enc error
fbNCErrorFFO(
    stMotionStage:=stMotionStage,
    fbFFHWO:=fbFFHWO,
    bAutoReset:=TRUE,
    nLowErrorId:=16#4500,
    nHighErrorId:=16#45FF,
);
fbEncErrorFFO(
    stMotionStage:=stMotionStage,
    fbFFHWO:=fbFFHWO,
    bAutoReset:=TRUE,
);
// Fast fault output is TRUE when there are no issues and FALSE when there is an issue
fbFFHWO.EvaluateOutput();

TestNC(0);
TestEnc(1);

IF bOneTestDone THEN
    bOneTestDone := FALSE;
    nTestCounter := nTestCounter + 1;
    tonTimer(IN:=FALSE);
    fbCauseNCError(
        Axis:=stMotionStage.Axis,
        bExecute:=FALSE,
    );
    stMotionStage.bReset := TRUE;
    fbMotionStage(stMotionStage:=stMotionStage);
END_IF
// Use this timer to time out any tests that stall
tonTimer(
    IN:=TRUE,
    PT:=T#5s,
);

METHOD TestEnc
VAR_INPUT
    nTestID: UINT;
END_VAR
VAR_INST
    nState: UINT;
END_VAR

TEST('TestEncError');
IF nTestCounter <> nTestID THEN
    RETURN;
END_IF

CASE nState OF
    0:
        // First cycle: no error, no fault
        AssertFalse(
            stMotionStage.bError,
            'Should have had no error before running this test',
        );
        AssertTrue(
            fbFFHWO.q_xFastFaultOut,
            'Should have had no fault with no error',
        );
        nState := 1;
    1:
        // Next time: cause an error
        fbCauseNCError(
            Axis:=stMotionStage.Axis,
            bExecute:=TRUE,
            nErrorCode:=16#4467, // Invalid encoder position data
        );
END_CASE

// Wait for the fault or the timeout, then check everything
IF tonTimer.Q OR (NOT fbFFHWO.q_xFastFaultOut AND stMotionStage.nErrorID = 16#4467) THEN
    AssertFalse(
        tonTimer.Q,
        'Timeout in test',
    );
    AssertTrue(
        stMotionStage.bError,
        'Did not get motor error in error test',
    );
    AssertEquals_UDINT(
        Expected:=16#4467,
        Actual:=stMotionStage.nErrorId,
        Message:='Error causer is broken',
    );
    AssertFalse(
        fbFFHWO.q_xFastFaultOut,
        Message:='Did not cause a fast fault',
    );
    AssertFalse(
        fbNCErrorFFO.bTripped,
        Message:='Drive error FB tripped with an enc error',
    );
    AssertTrue(
        fbEncErrorFFO.bTripped,
        Message:='Enc error fb did not trip with an enc error',
    );
    bOneTestDone := TRUE;
    nState := 0;
    TEST_FINISHED();
END_IF
END_METHOD

METHOD TestNC
VAR_INPUT
    nTestID: UINT;
END_VAR
VAR_INST
    nState: UINT;
END_VAR

TEST('TestNCError');
IF nTestCounter <> nTestID THEN
    RETURN;
END_IF

CASE nState OF
    0:
        // First cycle: no error, no fault
        AssertFalse(
            stMotionStage.bError,
            'Should have had no error before running this test',
        );
        AssertTrue(
            fbFFHWO.q_xFastFaultOut,
            'Should have had no fault with no error',
        );
        nState := 1;
    1:
        // Next time: cause an error
        fbCauseNCError(
            Axis:=stMotionStage.Axis,
            bExecute:=TRUE,
            nErrorCode:=16#4550, // Position lag monitoring error code
        );
END_CASE

// Wait for the fault or the timeout, then check everything
IF tonTimer.Q OR (NOT fbFFHWO.q_xFastFaultOut AND stMotionStage.nErrorId = 16#4550) THEN
    AssertFalse(
        tonTimer.Q,
        'Timeout in test',
    );
    AssertTrue(
        stMotionStage.bError,
        'Did not get motor error in error test',
    );
    AssertEquals_UDINT(
        Expected:=16#4550,
        Actual:=stMotionStage.nErrorId,
        Message:='Error causer is broken',
    );
    AssertFalse(
        fbFFHWO.q_xFastFaultOut,
        Message:='Did not cause a fast fault',
    );
    AssertTrue(
        fbNCErrorFFO.bTripped,
        Message:='NC error FB did not trip with a drive error',
    );
    AssertFalse(
        fbEncErrorFFO.bTripped,
        Message:='Enc error tripped with a drive error',
    );
    bOneTestDone := TRUE;
    TEST_FINISHED();
END_IF
END_METHOD

END_FUNCTION_BLOCK

// Tests/FB_PerMotorFFOND_Test
FUNCTION_BLOCK FB_PerMotorFFOND_Test EXTENDS TcUnit.FB_TestSuite
(*
    FFO if an illogical motor count is passed
    FFO if any motor has what looks like an encoder error
       - We'll just simulate this without doing it legit
       - The legit test is done elsewhere
    More FFOs may be added later and these will need to be tested too
*)
VAR
END_VAR


TestBlankCount();
TestTwoMotorEncError();

METHOD TestBlankCount : BOOL
VAR_INST
    fbFFO: FB_PerMotorFFOND;
    astMotionStage: ARRAY[1..MotionConstants.MAX_STATE_MOTORS] OF ST_MotionStage;
    fbFFHWO: FB_HardwareFFOutput := (bAutoReset := TRUE);
END_VAR

TEST('TestBlankCount');

fbFFHWO.EvaluateOutput();
AssertTrue(
    fbFFHWO.q_xFastFaultOut,
    'Started with a fault',
);
fbFFO(
    astMotionStage:=astMotionStage,
    fbFFHWO:=fbFFHWO,
);
fbFFHWO.EvaluateOutput();
AssertFalse(
    fbFFHWO.q_xFastFaultOut,
    'Blank count did not fault',
);
AssertTrue(
    fbFFO.bMotorCountError,
    'Blank count did not error',
);

TEST_FINISHED();
END_METHOD

METHOD TestTwoMotorEncError : BOOL
VAR_INST
    fbFFO: FB_PerMotorFFOND;
    astMotionStage: ARRAY[1..MotionConstants.MAX_STATE_MOTORS] OF ST_MotionStage;
    fbFFHWO: FB_HardwareFFOutput := (bAutoReset := TRUE);
END_VAR

TEST('TestTwoMotorEncError');

fbFFHWO.EvaluateOutput();
AssertTrue(
    fbFFHWO.q_xFastFaultOut,
    'Started with a fault',
);
astMotionStage[2].bError := TRUE;
astMotionStage[2].nErrorId := 16#4467; // Invalid encoder position data
fbFFO(
    astMotionStage:=astMotionStage,
    fbFFHWO:=fbFFHWO,
    nActiveMotorCount:=2,
);
fbFFHWO.EvaluateOutput();
AssertFalse(
    fbFFHWO.q_xFastFaultOut,
    'Encoder error did not fault',
);

TEST_FINISHED();
END_METHOD

END_FUNCTION_BLOCK

// Tests/FB_PositionStateMove_Test
FUNCTION_BLOCK FB_PositionStateMove_Test EXTENDS FB_MotorTestSuite
(*
    Test that FB_PositionStateMove can be used to move motors to named state positions
    And that the API behaves exactly as described.
*)
VAR
    stMotionStage: ST_MotionStage;
    fbMotionStage: FB_MotionStage;
    astPositionState: ARRAY[1..GeneralConstants.MAX_STATES] OF ST_PositionState;
    afbInternal: ARRAY[1..3] OF FB_PositionStateInternal;
    stDummyPos: ST_PositionState;
    stInvalid: ST_PositionState;
    stNotUpdated: ST_PositionState;
    stUnsafe: ST_PositionState;
    fbMove: FB_PositionStateMove;

    nTestCounter: UINT;
    bOneTestDone: BOOL;
    fTestStartPos: LREAL;
    tonTimer: TON;
    tonCleanup: TON;
    nIter: DINT;
    bStatesReady: BOOL;
END_VAR


astPositionState[1].sName := 'UNO';
astPositionState[1].fPosition := 10;
astPositionState[1].fDelta := 1;
astPositionState[1].fVelocity := 10;
SetGoodState(astPositionState[1]);

astPositionState[2].sName := 'DOS';
astPositionState[2].fPosition := 20;
astPositionState[2].fDelta := 1;
astPositionState[2].fVelocity := 10;
SetGoodState(astPositionState[2]);

astPositionState[3].sName := 'TRES';
astPositionState[3].fPosition := 30;
astPositionState[3].fDelta := 1;
astPositionState[3].fVelocity := 10;
SetGoodState(astPositionState[3]);

bStatesReady := TRUE;
FOR nIter := 1 TO 3 DO
    afbInternal[nIter](
        stMotionStage:=stMotionStage,
        stPositionState:=astPositionState[nIter],
    );
    bStatesReady := bStatesReady AND astPositionState[nIter].bUpdated;
END_FOR
stInvalid.bValid := FALSE;
stInvalid.bUpdated := TRUE;
stInvalid.bMoveOk := TRUE;
stNotUpdated.bValid := TRUE;
stNotUpdated.bUpdated := FALSE;
stNotUpdated.bMoveOk := TRUE;
stUnsafe.bValid := TRUE;
stUnsafe.bUpdated := TRUE;
stUnsafe.bMoveOk := FALSE;

SetEnables(stMotionStage);
fbMotionStage(stMotionStage:=stMotionStage);

IF bStatesReady AND nTestCounter = 0 THEN
    // Don't run any tests until the states are ready
    nTestCounter := 1;
    // Warm up the motion FB with a exec false runthrough
    fbMove(
        stMotionStage:=stMotionStage,
        stPositionState:=stDummyPos,
        bExecute:=FALSE,
    );
END_IF

// Test that we can move to state 1 and the outputs are correct as we go
TestMove(1, 1, FALSE);
// Test that we can move to state 2 and the outputs are correct as we go
TestMove(2, 2, FALSE);
// Test that we can interrupt a move to state 3 by dropping bExecute
TestMove(3, 3, TRUE);
// Test that we cannot move to an invalid state
TestBadStates(4);
// Test that we need a new bExecute to start a new move if a move goes from unsafe to safe
TestMoveOk(5);

// Wait a few cycles for remaining errors to propagate
tonCleanup(IN:=bOneTestDone, PT:=T#1s);
IF tonCleanup.Q THEN
    IF fbMove.bBusy THEN
        fbMove(
            stMotionStage:=stMotionStage,
            stPositionState:=stDummyPos,
            bExecute:=FALSE,
            bReset:=FALSE,
        );
    ELSIF stMotionStage.bBusy THEN
        stMotionStage.bExecute := FALSE;
    ELSIF fbMove.bError THEN
        fbMove(
            stMotionStage:=stMotionStage,
            stPositionState:=stDummyPos,
            bExecute:=FALSE,
            bReset:=TRUE,
        );
    ELSIF stMotionStage.bError THEN
       stMotionStage.bReset := TRUE;
    ELSE
        fbMove(
            stMotionStage:=stMotionStage,
            stPositionState:=stDummyPos,
            bExecute:=FALSE,
            bReset:=FALSE,
        );
        stMotionStage.bReset := FALSE;

        bOneTestDone := FALSE;
        nTestCounter := nTestCounter + 1;
        tonTimer(IN:=FALSE);
    END_IF
END_IF
// Use this timer to time out any tests that stall
tonTimer(
    IN:=bStatesReady,
    PT:=T#5s,
);

METHOD TestBadStates
VAR_INPUT
    nTestIndex: UINT;
END_VAR
TEST(CONCAT('TestInvalid', UINT_TO_STRING(nTestIndex)));
IF nTestCounter <> nTestIndex OR bOneTestDone THEN
    RETURN;
END_IF

AssertFalse(
    fbMove.bError,
    'Started with an error',
);

fbMove(
    stMotionStage:=stMotionstage,
    stPositionState:=stInvalid,
    bExecute:=TRUE,
);

AssertTrue(
    fbMove.bError,
    'Invalid should have given an error',
);

fbMove(
    stMotionStage:=stMotionstage,
    stPositionState:=stInvalid,
    bExecute:=FALSE,
    bReset:=TRUE,
);

AssertFalse(
    fbMove.bError,
    'Started with an error',
);

fbMove(
    stMotionStage:=stMotionstage,
    stPositionState:=stNotUpdated,
    bExecute:=TRUE,
    bReset:=FALSE,
);

AssertTrue(
    fbMove.bError,
    'Not updated should have given an error',
);

fbMove(
    stMotionStage:=stMotionstage,
    stPositionState:=stNotUpdated,
    bExecute:=FALSE,
    bReset:=TRUE,
);

AssertFalse(
    fbMove.bError,
    'Started with an error',
);

fbMove(
    stMotionStage:=stMotionstage,
    stPositionState:=stUnsafe,
    bExecute:=TRUE,
    bReset:=FALSE,
);

AssertTrue(
    fbMove.bError,
    'Unsafe should have given an error',
);

bOneTestDone := TRUE;
TEST_FINISHED();
END_METHOD

METHOD TestMove
VAR_INPUT
    nTestIndex: UINT;
    nStateIndex: UINT;
    bInterrupt: BOOL;
END_VAR
VAR_INST
    bLocalInit: BOOL;
    bInterruptStarted: BOOL;
    tonBusy: TON;
END_VAR
TEST(CONCAT('TestMove', UINT_TO_STRING(nTestIndex)));
IF nTestCounter <> nTestIndex OR bOneTestDone THEN
    RETURN;
END_IF

IF NOT bLocalInit THEN
    // Starting output checks
    AssertFalse(
        Condition:=fbMove.bBusy,
        Message:='Tried to start test with busy motor',
    );
    AssertFalse(
        Condition:=fbMove.bError,
        Message:='Tried to start test with errored motor',
    );
    bLocalInit := TRUE;
END_IF

// Simulate waiting a moment before stopping
tonBusy(IN:=stMotionStage.bBusy, PT:=T#100ms);
bInterruptStarted S= bInterrupt AND tonBusy.Q;

fbMove(
    stMotionStage:=stMotionstage,
    stPositionState:=astPositionState[nStateIndex],
    bExecute:=NOT bInterruptStarted,
);

IF fbMove.bDone OR tonTimer.Q OR (bInterruptStarted AND NOT fbMove.bBusy) THEN
    AssertFalse(
        tonTimer.Q,
        'Test timed out',
    );
    IF bInterrupt THEN
        AssertFalse(
            fbMove.bAtState,
            Message:='Should have been interrupted, but made it to the goal',
        );
    ELSE
        AssertTrue(
            fbMove.bAtState,
            Message:='Did not end at the state',
        );
        AssertEquals_LREAL(
            Expected:=astPositionState[nStateIndex].fPosition,
            Actual:=stMotionStage.stAxisStatus.fActPosition,
            Delta:=0.01,
            Message:='Did not reach the goal state',
        );
    END_IF
    AssertFalse(
        fbMove.bBusy,
        Message:='Was busy while done',
    );
    AssertFalse(
        fbMove.bError,
        Message:=CONCAT('Should not end in error: ', stMotionStage.sErrorMessage),
    );

    bOneTestDone := TRUE;
    bLocalInit := FALSE;
    bInterruptStarted := FALSE;
    TEST_FINISHED();
END_IF
END_METHOD

METHOD TestMoveOk
VAR_INPUT
    nTestIndex: UINT;
END_VAR
VAR_INST
    nStep: UINT;
    fStartPos: LREAL;
    stState: ST_PositionState := (
        sName:='GOAL',
        fPosition:=135,
        fDelta:=0.5,
        fVelocity:=1,
        bValid:=TRUE,
        bMoveOk:=FALSE,
        bUpdated:=TRUE
    );
    tonInternal: TON;
    bLocalExec: BOOL;
    bLocalReset: BOOL;
END_VAR
VAR CONSTANT
    END: UINT := 999;
END_VAR
TEST('TestMoveOk');
IF nTestCounter <> nTestIndex OR bOneTestDone THEN
    RETURN;
END_IF

CASE nStep OF
    // Initial setup and checks
    0:
        fStartPos := stMotionStage.stAxisStatus.fActPosition;
        AssertFalse(
            fbMove.bError,
            'Started with a fbMove error',
        );
        AssertFalse(
            stMotionStage.bError,
            'Started with a motor error',
        );
        bLocalExec := FALSE;
        bLocalReset := FALSE;
        nStep := nStep + 1;
    // Move to a state that is bad
    1:
        stState.bMoveOk := FALSE;
        bLocalExec := TRUE;
        nStep := nStep + 1;
    // The move should have failed with an error on the FB that never propagated to the motor itself- we shouldn't have attempted the move at all
    2:
        AssertTrue(
            fbMove.bError,
            'Did not have the expected move not ok error',
        );
        AssertFalse(
            stMotionStage.bError,
            'Had a motion error, but we never should have asked for a move?',
        );
        nStep := nStep + 1;
    // Make the state no longer bad, and wait a bit
    3:
        stState.bMoveOk := TRUE;
        tonInternal(IN:=TRUE, PT:=T#500ms);
        IF tonInternal.Q THEN
            tonInternal(IN:=FALSE);
            nStep := nStep + 1;
        END_IF
    // There should be no movement still
    4:
        AssertEquals_LREAL(
            Expected:=fStartPos,
            Actual:=stMotionStage.stAxisStatus.fActPosition,
            Delta:=0.1,
            Message:='Motor moved without bReset or a new bExecute!',
        );
        // Reset the error (rising edge)
        bLocalReset := TRUE;
        nStep := nStep + 1;
    // After we reset the error, wait a bit
    5:
        // Drop for rising edges later
        bLocalReset := FALSE;
        tonInternal(IN:=TRUE, PT:=T#500ms);
        IF tonInternal.Q THEN
            tonInternal(IN:=FALSE);
            nStep := nStep + 1;
        END_IF
    // There should be no error, and STILL be no movement
    6:
        AssertFalse(
            fbMove.bError,
            'The error should be reset',
        );
        AssertEquals_LREAL(
            Expected:=fStartPos,
            Actual:=stMotionStage.stAxisStatus.fActPosition,
            Delta:=0.1,
            Message:='Motor moved without a new bExecute!',
        );
        // Set bExecute to FALSE for an upcoming rising edge. It should be TRUE at this point.
        bLocalExec := FALSE;
        nStep := nStep + 1;
    // We should be able to start a move via bExecute now
    7:
        stState.fVelocity := 2000;
        stState.fAccel := 15000;
        stState.fDecel := 15000;
        bLocalExec := TRUE;
        IF fbMove.bAtState AND stMotionStage.bDone THEN
            nStep := END;
        END_IF
END_CASE

// Run fbMove exactly once every cycle no matter what
fbMove(
    stMotionStage:=stMotionStage,
    stPositionState:=stState,
    bExecute:=bLocalExec,
    bReset:=bLocalReset,
);

IF nStep = END OR tonTimer.Q THEN
    AssertFalse(
        tonTimer.Q,
        'Test timed out',
    );
    // Check that we've reached the goal
    AssertEquals_LREAL(
        Expected:=stState.fPosition,
        Actual:=stMotionStage.stAxisStatus.fActPosition,
        Delta:=0.1,
        Message:='Motor did not reach the goal.',
    );
    bOneTestDone := TRUE;
    TEST_FINISHED();
END_IF
END_METHOD

END_FUNCTION_BLOCK

// Tests/FB_PositionStateMoveND_Test
FUNCTION_BLOCK FB_PositionStateMoveND_Test EXTENDS FB_MotorTestSuite
(*
    Test that FB_PositionStateMoveND can be used to move motors to named state positions
    And that the API behaves exactly as described.
*)
VAR
    astMotionStage: ARRAY[1..MotionConstants.MAX_STATE_MOTORS] OF ST_MotionStage;
    afbMotionStage: ARRAY[1..3] OF FB_MotionStage;
    astGoalPositions: ARRAY[1..MotionConstants.MAX_STATE_MOTORS] OF ST_PositionState;
    afbInternal: ARRAY[1..3] OF FB_PositionStateInternal;
    stDummyPos: ST_PositionState;
    fbMove: FB_PositionStateMoveND;

    bInit: BOOL;
    nTestCounter: UINT;
    bOneTestDone: BOOL;
    fTestStartPos: LREAL;
    tonTimer: TON;
    nIter: DINT;
    bStatesReady: BOOL;
END_VAR


IF NOT bInit THEN
    ResetGoals();
    bInit := TRUE;
END_IF

bStatesReady := TRUE;
FOR nIter := 1 TO 3 DO
    afbInternal[nIter](
        stMotionStage:=astMotionStage[nIter],
        stPositionState:=astGoalPositions[nIter],
    );
    bStatesReady := bStatesReady AND astGoalPositions[nIter].bUpdated;
    SetEnables(astMotionStage[nIter]);
    afbMotionStage[nIter](stMotionStage:=astMotionStage[nIter]);
END_FOR

IF bStatesReady AND nTestCounter = 0 THEN
    // Don't run any tests until the states are ready
    nTestCounter := 1;
    // Warm up the motion FB with a exec false runthrough
    fbMove(
        astMotionStage := astMotionStage,
        astPositionState := astGoalPositions,
        nActiveMotorCount := 3,
        bExecute := FALSE,
    );
END_IF

// Move to somewhere
TestMove(1, 1, 5, 10, FALSE);
// Somewhere else
TestMove(2, -10, 0, 5, FALSE);
// Interrupt on the way to the last place
TestMove(3, 0, 0, 0, TRUE);

IF bOneTestDone THEN
    bOneTestDone := FALSE;
    nTestCounter := nTestCounter + 1;
    ResetGoals();
    fbMove(
        astMotionStage := astMotionStage,
        astPositionState := astGoalPositions,
        nActiveMotorCount := 3,
        bExecute := FALSE,
        bReset := TRUE,
    );
    tonTimer(IN:=FALSE);
END_IF
// Use this timer to time out any tests that stall
tonTimer(
    IN:=bStatesReady,
    PT:=T#5s,
);

METHOD ResetGoals
VAR_INPUT
END_VAR

astGoalPositions[1].sName := 'Goal1';
astGoalPositions[1].fPosition := 0;
astGoalPositions[1].fDelta := 1;
astGoalPositions[1].fVelocity := 10;
astGoalPositions[1].bUseRawCounts := FALSE;
SetGoodState(astGoalPositions[1]);

astGoalPositions[2].sName := 'Goal2';
astGoalPositions[2].fPosition := 0;
astGoalPositions[2].fDelta := 1;
astGoalPositions[2].fVelocity := 10;
astGoalPositions[2].bUseRawCounts := FALSE;
SetGoodState(astGoalPositions[2]);

astGoalPositions[3].sName := 'Goal3';
astGoalPositions[3].fPosition := 0;
astGoalPositions[3].fDelta := 1;
astGoalPositions[3].fVelocity := 10;
astGoalPositions[3].bUseRawCounts := FALSE;
SetGoodState(astGoalPositions[3]);
END_METHOD

METHOD TestMove
VAR_INPUT
    nTestIndex: UINT;
    fMotor1Pos: LREAL;
    fMotor2Pos: LREAL;
    fMotor3Pos: LREAL;
    bInterrupt: BOOL;
END_VAR
VAR_INST
    bLocalInit: BOOL;
    bInterruptStarted: BOOL;
END_VAR
TEST(CONCAT('TestMove', UINT_TO_STRING(nTestIndex)));
IF nTestCounter <> nTestIndex THEN
    RETURN;
END_IF

IF NOT bLocalInit THEN
    // Starting output checks
    AssertFalse(
        Condition:=fbMove.bBusy,
        Message:='Tried to start test with busy motor',
    );
    AssertFalse(
        Condition:=fbMove.bError,
        Message:='Tried to start test with errored motor',
    );
    bLocalInit := TRUE;
END_IF

astGoalPositions[1].fPosition := fMotor1Pos;
astGoalPositions[2].fPosition := fMotor2Pos;
astGoalPositions[3].fPosition := fMotor3Pos;

bInterruptStarted S= bInterrupt AND astMotionStage[1].bBusy AND astMotionStage[2].bBusy AND astMotionStage[3].bBusy;
fbMove(
    astMotionStage:=astMotionStage,
    astPositionState:=astGoalPositions,
    nActiveMotorCount:=3,
    bExecute:=NOT bInterruptStarted,
);
IF fbMove.bDone OR tonTimer.Q OR (bInterruptStarted AND NOT fbMove.bBusy) THEN
    IF bInterrupt THEN
        AssertFalse(
            fbMove.bAtState,
            Message:='Should have been interrupted, but made it to the goal',
        );
    ELSE
        AssertTrue(
            fbMove.bAtState,
            Message:='Did not end at the state',
        );
        FOR nIter := 1 TO 3 DO
            AssertEquals_LREAL(
                Expected:=astGoalPositions[nIter].fPosition,
                Actual:=astMotionStage[nIter].stAxisStatus.fActPosition,
                Delta:=0.01,
                Message:='Did not reach the goal state',
            );
        END_FOR

    END_IF
    AssertFalse(
        fbMove.bBusy,
        Message:='Was busy while done',
    );
    AssertFalse(
        fbMove.bError,
        Message:='Should not end in error',
    );

    bOneTestDone := TRUE;
    TEST_FINISHED();
END_IF
END_METHOD

END_FUNCTION_BLOCK

// Tests/FB_PositionStateND_Test
FUNCTION_BLOCK FB_PositionStateND_Test EXTENDS FB_MotorTestSuite
(*
    Sanity checks for the following:
    - FB_PositionState1D
    - FB_PositionState2D
    - FB_PositionState3D
    The internals have already been tested, but we need to make sure that
    they've been put together at least somewhat sensibly.
    This FB will simply use each FB to move and check the results.

